(* CoDeSys 2.3 project: cy-22-wg-005.pro *)
(* Title: cy-22-wg - ClevergyAS *)
(* Libraries: Standard.lib 2.12.10 14:48:34, Util.lib 26.9.14 10:12:46, Visual.lib 2.12.10 14:48:34, WagoLibIdent.lib 25.2.13 11:12:16, WagoLibStatus.lib 2.12.10 14:48:32, SysLibFile.lib 2.12.10 14:48:34, SysLibRtc.lib 2.12.10 14:48:32, SysLibSockets.lib 10.2.11 09:20:54, SysLibEvent.lib 2.12.10 14:48:34, SysLibPlcCtrl.lib 2.12.10 14:48:32, SysLibCallback.lib 2.12.10 14:48:32, mod_com.lib 2.12.10 14:48:32, SerComm.lib 31.5.11 08:54:36, Serial_Interface_01.lib 22.4.13 12:50:14, Modb_l05.lib 22.4.13 12:50:12, WagoLibModbus_IP_01.lib 24.7.13 15:05:58 *)

(* PLC configuration (modules and I/O channels)
VPN_OUT2 AT %IX6.0 [BOOLOnX_I] Ch_1 Digital input
KEY_QE_ST AT %IX6.1 [BOOLOnX_I] Ch_2 Digital input
SCA01_1_DI AT %IX6.2 [BOOLOnX_I] Ch_3 Digital input
SCA01_2_DI AT %IX6.3 [BOOLOnX_I] Ch_4 Digital input
SCA01_3_DI AT %IX6.4 [BOOLOnX_I] Ch_5 Digital input
AT %IX6.5 [BOOLOnX_I] Ch_6 Digital input
AT %IX6.6 [BOOLOnX_I] Ch_7 Digital input
AT %IX6.7 [BOOLOnX_I] Ch_8 Digital input
DIG_TA1 AT %IW0 [WORDOnW_I] Ch_1 Input word
DIG_TA2 AT %IW1 [WORDOnW_I] Ch_2 Input word
0750-0653/0003-0000#03 RS485 Interface (Adjustable), 3 Bytes [Type_21_1_Channels] node 2, in %IB8 out %QB4 {INTTypePAAssignment = PLC; INTTypeModule = plugged}
  AT %IX2.0 [BOOLOnX_I] Transmission acknowledgement
  AT %IX2.1 [BOOLOnX_I] Reception request
  AT %IX2.2 [BOOLOnX_I] Initialization acknowledgement
  AT %IX2.3 [BOOLOnX_I] Input buffer is full
  AT %IX2.4 [BOOLOnX_I] Number of received characters Bit 0
  AT %IX2.5 [BOOLOnX_I] Number of received characters Bit 1
  AT %IX2.6 [BOOLOnX_I] Number of received characters Bit 2
  AT %IB5 [BYTEOnB_I] Input data Byte 0
  AT %IB6 [BYTEOnB_I] Input data Byte 1
  AT %IB7 [BYTEOnB_I] Input data Byte 2
  AT %QX0.0 [BOOLOnX_Q] Transmission request
  AT %QX0.1 [BOOLOnX_Q] Reception acknowledgement
  AT %QX0.2 [BOOLOnX_Q] Initialization request
  AT %QX0.4 [BOOLOnX_Q] Number of characters Bit 0
  AT %QX0.5 [BOOLOnX_Q] Number of characters Bit 1
  AT %QX0.6 [BOOLOnX_Q] Number of characters Bit 2
  AT %QB1 [BYTEOnB_Q] Output data Byte 0
  AT %QB2 [BYTEOnB_Q] Output data Byte 1
  AT %QB3 [BYTEOnB_Q] Output data Byte 2
0750-0653/0003-0000#03 RS485 Interface (Adjustable), 3 Bytes [Type_21_1_Channels] node 3, in %IB12 out %QB4 {INTTypePAAssignment = PLC; INTTypeModule = plugged}
  AT %IX4.0 [BOOLOnX_I] Transmission acknowledgement
  AT %IX4.1 [BOOLOnX_I] Reception request
  AT %IX4.2 [BOOLOnX_I] Initialization acknowledgement
  AT %IX4.3 [BOOLOnX_I] Input buffer is full
  AT %IX4.4 [BOOLOnX_I] Number of received characters Bit 0
  AT %IX4.5 [BOOLOnX_I] Number of received characters Bit 1
  AT %IX4.6 [BOOLOnX_I] Number of received characters Bit 2
  AT %IB9 [BYTEOnB_I] Input data Byte 0
  AT %IB10 [BYTEOnB_I] Input data Byte 1
  AT %IB11 [BYTEOnB_I] Input data Byte 2
  AT %QX2.0 [BOOLOnX_Q] Transmission request
  AT %QX2.1 [BOOLOnX_Q] Reception acknowledgement
  AT %QX2.2 [BOOLOnX_Q] Initialization request
  AT %QX2.4 [BOOLOnX_Q] Number of characters Bit 0
  AT %QX2.5 [BOOLOnX_Q] Number of characters Bit 1
  AT %QX2.6 [BOOLOnX_Q] Number of characters Bit 2
  AT %QB5 [BYTEOnB_Q] Output data Byte 0
  AT %QB6 [BYTEOnB_Q] Output data Byte 1
  AT %QB7 [BYTEOnB_Q] Output data Byte 2
LUX5_EN AT %QX4.0 [BOOLOnX_Q] Ch_1 Digital output
LUX6_EN AT %QX4.1 [BOOLOnX_Q] Ch_2 Digital output
LUX3_EN AT %QX4.2 [BOOLOnX_Q] Ch_1 Digital output
LUX4_EN AT %QX4.3 [BOOLOnX_Q] Ch_2 Digital output
LUX1_EN AT %QX4.4 [BOOLOnX_Q] Ch_1 Digital output
LUX2_EN AT %QX4.5 [BOOLOnX_Q] Ch_2 Digital output
Fieldbus variables [FB_VARS] node 1, in %IB0 out %QB0
Flag variables [FLAG_VARS] node 2, in %IB0 out %QB0
Modbus-Master [MB_MASTER] node 3, in %IB0 out %QB0
*)

(* Global variable list: Global_Constants *)
VAR_GLOBAL CONSTANT

	Plant_NAME			: STRING :='cySN:22 cyVER:0 - Coin OVS Curno';
	Plant_SN			: DWORD  :=22;	  	(* S/N Impianto di telecontrollo *)
	Plant_SW_VER		: WORD   :=0;		(* Versione SW installata *)

	(* Colour defines *)
	COLOR_RED			: DWORD	:= 16#2020F0;
	COLOR_YELLOW		: DWORD	:= 16#20F0F0;
	COLOR_GREEN			: DWORD	:= 16#20F020;
	COLOR_GREEN_OFF		: DWORD := 16#006000;

	(* Parameters *)
	Plant_DefaultTAmb	: INT	:=100;		(* [.1°C] Temperatura ambiente di default in caso di rottura sonda *)
	Plant_MaxRunTAmb	: INT   :=250; 		(* [.1°C] Temperatura ambiente massima funzionamento impianto *)
	Plant_AntiFreezeTAmb: INT   :=-40;		(* [.1°C] Antifreeze temperature, start circulators *)
	Plant_VRD_TAlarm	: INT   :=450; 		(* [.1°C] Temperatura di allarme VRD, blocco *)
	Plant_VRD_TMax		: INT   :=430; 		(* [.1°C] Setpoint massimo per uscita VRD *)
	Plant_VRD_TDefault	: INT	:=300;		(* [.1°C] Temperatura di default in caso di errore climatica *)
	Plant_CirOffDelay	: TIME	:=T#15m;	(* (Def.T#15m) Ritardo spegnimento pompe per ricircolo caldaia *)
	Plant_MaxWaterLoss	: WORD  :=2;		(* [lt/h] Massima perdita del circuito *)

	FeedbackTolerance	: WORD	:= 5;		(* 10% Tolerance on read measures *)

	(* Filesystem *)
	FilesPath  			: STRING :='S:\';

	(* TCP Logger *)
	Logger_SERVER		: STRING:='';
	Logger_IP			: STRING:='192.168.100.3';
	Logger_PORT			: WORD  :=80;
	Logger_GETSTART		: STRING:='GET /cygmsrv/hsgm.ashx?';
	Logger_GETEND		: STRING:='$R$N$R$N';
	Logger_CHECK		: STRING:='True';
	Logger_CRLF			: STRING:='$R$N';
	Logger_DataFile		: STRING:='S:\LOG.DAT';
	Logger_DataFileOld	: STRING:='S:\LOG.BCK';
	Logger_IndexFile	: STRING:='S:\LOG.IDX';
	Logger_ConnRetries	: BYTE:=5;
	Logger_RecoverMsgs	: BYTE:=25;

	(* TCP Remote *)
	Remote_PORT			: WORD  :=10;
	Remote_WELCOME		: STRING:='Connected$R$N';
	Remote_OK			: STRING:='OK$R$N';
	Remote_ERROR		: STRING:='ERROR$R$N';

	(* TCP Sockets *)
	MAX_SEND_TCP_SERVER					 : DWORD:=3000;(*60000*)
	MAX_RECEIVE_TCP_SERVER				 : DWORD:=3000;
	MAX_RECEIVE_TCP_SERVER_SOCKET	 	 : DWORD:=1500;
	MAX_SEND_TCP_CLIENT					 : DWORD:=3000;(*15000*)
	MAX_RECEIVE_TCP_CLIENT				 : DWORD:=1500;
	MAX_RECEIVE_TCP_CLIENT_SOCKET		 : DWORD:=1500;
	MAX_RECEIVE_UDP_SERVER				 : INT  :=1472;
	MAX_RECEIVE_UDP_CLIENT				 : INT  :=1472;
	CONNECT_WATCHDOG_TIME				 : TIME :=t#10s;

END_VAR

(* Global variable list: Global_Retain *)
VAR_GLOBAL RETAIN PERSISTENT
	Mode_Manual : BOOL := FALSE;

	Lux_ref	:	ARRAY [1..2,1..7] OF WORD;

	LuxWT	:	ARRAY [1..6] OF DWORD;	(* Lux working time non volatile counters *)
	LuxPOC	:	ARRAY [1..6] OF DWORD;	(* Lux power on cycles non volatile counters *)
END_VAR

(* Global variable list: Global_Variables *)
VAR_GLOBAL

	SYS    : typ_SYS;
	Logger : typ_Logger;
	CronEd : obj_CRON_EDITOR;

	(**** PLANT OBJECTS ****)
	CRON01 : obj_CRON		:= ( ID:=1 );		(* Controllo LUX01 *)
	CRON02 : obj_CRON		:= ( ID:=2 );		(* Controllo LUX02 *)
	CRON03 : obj_CRON		:= ( ID:=3 );		(* Controllo LUX03 *)
	CRON04 : obj_CRON		:= ( ID:=4 );		(* Controllo LUX04 *)
	CRON05 : obj_CRON		:= ( ID:=5 );		(* HVAC01 - Start Stop  *)
	CRON06 : obj_CRON		:= ( ID:=6 );		(* HVAC01 - Set Point raffreddamento *)
	CRON07 : obj_CRON		:= ( ID:=7 );		(* HVAC01 - Set Point riscaldamento *)
	CRON08 : obj_CRON		:= ( ID:=8 );		(* HVAC01 - ??? Set Point ECO Soglia Minima *)
	CRON09 : obj_CRON		:= ( ID:=9 );		(* HVAC01 - ??? Set Point ECO Soglia Massima *)
	CRON10 : obj_CRON		:= ( ID:=10 );		(* HVAC02 - Start Stop *)
	CRON11 : obj_CRON		:= ( ID:=11 );		(* HVAC02 - Set Point raffreddamento *)
	CRON12 : obj_CRON		:= ( ID:=12 );		(* HVAC02 - Set Point riscaldamento *)
	CRON13 : obj_CRON		:= ( ID:=13 );		(* HVAC02 - ??? Set Point ECO Soglia Minima *)
	CRON14 : obj_CRON		:= ( ID:=14 );		(* HVAC02 - ??? Set Point ECO Soglia Massima *)

	LUX01  : obj_LUXP		:= ( ID:=1, CTRL_MODE:=2, KEY_DEV:=FALSE );		(* Control mode: Scheduled -> Crono	*)
	LUX02  : obj_LUXP		:= ( ID:=2, CTRL_MODE:=2 );		(* Control mode: Scheduled -> Crono	*)
	LUX03  : obj_LUXP		:= ( ID:=3, CTRL_MODE:=0, KEY_DEV:=TRUE );		(* Control mode: Manual -> Switch *)
	LUX04  : obj_LUXP		:= ( ID:=4, CTRL_MODE:=2 );		(* Control mode: Scheduled -> Crono	*)
	LUX05  : obj_LUXP		:= ( ID:=5, CTRL_MODE:=2 );		(* Control mode: Scheduled -> Crono	*)
	LUX06  : obj_LUXP		:= ( ID:=6, CTRL_MODE:=1 );		(* Control mode: Automatic -> External device/sensor	*)

	AID01  : obj_ANALOG_IN_DIFF				:= (ID:=1, Lines:=3);
	AID02  : obj_ANALOG_IN_DIFF				:= (ID:=2, Lines:=3);

	MODB01 : obj_MODBUS						:= ( ID:=1 , COM:=2, BAUDRATE:=BAUD_9600, RS485:=TRUE );
	ANZ01  : obj_MODBUS_FRER_QUBOH			:= ( ID:=1 , Address:=1 );
	ANZ02  : obj_MODBUS_FRER_QUBOH			:= ( ID:=2 , Address:=2 );

	MODB02 : obj_MODBUS						:= ( ID:=2 , COM:=3, BAUDRATE:=BAUD_9600, RS485:=TRUE );
	HVAC01 : obj_HVAC_LENNOX_FGK190H2M_new	:= ( ID:=1 , ADDRESS:=1 );
	HVAC02 : obj_HVAC_LENNOX_FGK190H2M_new	:= ( ID:=2 , ADDRESS:=2 );

	MODB03 : obj_MODBUS_TCP					:= ( ID:=1,IP:='192.168.100.11');
	ZTHL01 : obj_ZTHL						:= ( ID:=1, Address:=2);
	ZTHL02 : obj_ZTHL						:= ( ID:=2, Address:=3);
	ZTHL03 : obj_ZTHL						:= ( ID:=3, Address:=5);
	ZTHL04 : obj_ZTHL						:= ( ID:=4, Address:=6);

	(**** SIMULATION ONLY ****)
(*	VPN_ST2		:BOOL:=TRUE;
	KEY_QE_ST	:BOOL:=TRUE;
*)

END_VAR

(* Data type in Logger *)
TYPE en_Logger_ErrLev :
(
	EL_Log			:=0,
	EL_Wrn			:=1,
	EL_Alarm			:=2,
	EL_AlarmStop		:=3
);
END_TYPE

(* Data type in Logger *)
TYPE en_Logger_Status :
(
	S_Logger_UNKNOWN := 0,
	S_Logger_IDLE,
	S_Logger_WAITCONN,
	S_Logger_WAITTX,
	S_Logger_WAITRESP,
	S_Logger_ERROR
);
END_TYPE

(* Data type *)
TYPE en_SYS_Objects :
(
	EO_SYS		:=0,  (* PLC *)
	EO_VPN		:=1,  (* VPN *)
	EO_DOOR	:=2,  (* Door & access control *)

	EO_CAL		:=10, (* Caldaia *)
	EO_CIR		:=11, (* Circolatore *)
	EO_CRON		:=12, (* Crono-termostato *)
	EO_VRD		:=13, (* Valvola miscelatore pannelli *)
	EO_CTL		:=14, (* Contalitri *)
	EO_CTB		:=15, (* Contabilizzatore *)
	EO_TPV		:=16, (* Temperature probes values *)
	EO_PPV		:=17, (* Pressure probes values *)
	EO_PBV		:=18, (* Over-Pressure Alarms *)
	EO_TBV		:=19, (* Over-Temperature Alarms *)
	EO_PMV		:=20, (* Under-Pressure Alarms *)
	EO_GRU		:=21, (* Gruppo termico *)
	EO_PDC		:=22, (* Pompa di calore *)
	EO_SOL		:=23, (* Pannello solare termico *)
	EO_ESOL		:=24, (* Pannello solare fotovoltaico *)
	EO_GAS		:=25, (* Contatore GAS *)
	EO_PORT		:=26, (* Misuratore di portata *)
	EO_FPV		:=27, (* Flow probes values *)
	EO_ANZ		:=28, (* Analizzatore di rete *)
	EO_SCA		:=29, (* Signal Control Alarms *)
	EO_LUX		:=30, (* Illumination point *)
	EO_LUXM		:=31, (* Metered illumination point*)
	EO_PSG		:=32, (* Sensore di passaggio *)
	EO_HVAC		:=33, (*Heating, Ventilating and Air Conditioning*)
	EO_HYGRV	:=34, (*Valori sensori di umidità relativa (0.1%)*)
	EO_COOV		:=35, (*Valori sensori CO2 (PPM)*)




	EO_ZGW			:=200,  (* ZigBee - Gateway *)
	EO_ZRM			:=201,	(* ZigBee - Repeater *)
	EO_ZREL			:=202,	(* ZigBee - Actuator rele *)
	EO_ZTHL			:=203,	(* ZigBee - Temperature Sensor *)

	EO_ASGW			:=250,	(* ASi - Gateway *)
	EO_ASCBI			:=251,	(* ASi - Input Board, Ciabatta *)

	EO_LON				:=1000, (* Bus - LON *)
	EO_MODBUS			:=1001, (* Bus - MODBUS *)
	EO_MBUS				:=1002, (* Bus - M-BUS *)
	EO_MODBUS_TCP	:=1003, (* Bus - MODBUS TCP *)

	EO_GENERIC			:=9000, (* Generic dataset *)
	EO_EXPO				:=9001 (* EXPO dataset *)
);
END_TYPE

(* Data type *)
TYPE en_SYS_Status :
(
	S_UNKNOWN  := 0,
	S_STARTUP,
	S_INIT_RTC,
	S_INIT_VAR,
	S_AUTOTEST,
	S_RUNNING,
	S_SHUTDOWN,
	S_HALT
);
END_TYPE

(* Data type in Plant_Objects *)
TYPE typ_Condition :
STRUCT
	Enable		:	BYTE;	(*	0: Condition event not used		(disable condition event)
								1: Boolean event: trig On	(rele, switch, sensors digital input..)
								2:    ''    ''  : trig Off		
								3:	  ''    ''  : trig On/Off
								4: Tod event: trig On		(Time of day)
								5: Tod event: trig Off		(Trig On/Off not expected -> it's a schedule! )
							 *)

	(* Boolean event *)
	OnIN		:	BOOL;	(* Input event generating an On *)
	OffIN		:	BOOL;	(* Input event generating an Off  *)

	OnValue		:	BOOL;	(* Value to trig an On *)
	OffValue	:	BOOL;	(*   ''        ''   Off	 *)


	(* Time of the day event (absolute time) *)
	OnTime		:	TOD;	(* Time at which trig an On (hh:mm) *)
	OffTime		:	TOD;	(*  ''            ''     Off (hh:mm)  *)


END_STRUCT
END_TYPE

(* Data type in Plant_Objects *)
TYPE typ_Cron_Calendar :
STRUCT
	Profile		: ARRAY[0..384] OF BYTE;
END_STRUCT
END_TYPE

(* Data type in Plant_Objects *)
TYPE typ_Cron_Jolly :
STRUCT
	Start		: DT;
	End			: DT;
	Temp		: WORD;
	Flags		: WORD; (* B0:Enabled B1..B15:Unused *)
END_STRUCT
END_TYPE

(* Data type in Plant_Objects *)
TYPE typ_Cron_Profile :
STRUCT
	Flags		: WORD;
	Setpoint	: ARRAY [0..95] OF WORD;
END_STRUCT
END_TYPE

(* Data type in Logger *)
TYPE typ_Logger :
STRUCT
	Status		: en_Logger_Status;

	SendReq		: BOOL;
	SendIdx		: DWORD;
	SendData	: ARRAY [0..MAX_SEND_TCP_CLIENT] OF BYTE;
	SendLen		: DINT;

	TData		: ARRAY [0..MAX_SEND_TCP_CLIENT] OF BYTE;
	TLen		: DINT;

	LastIdxPos	: DWORD;

	(* Temporary variables used by objects *)
	s1			: STRING(256);
	i1			: WORD;

END_STRUCT
END_TYPE

(* Data type in Plant_Objects *)
TYPE typ_MODBUS_ABB_DMTME72 :
STRUCT
	V_3P		: DWORD; (* V *)
	V_L1N		: DWORD;
	V_L2N		: DWORD;
	V_L3N		: DWORD;
	V_L1L2		: DWORD;
	V_L2L3		: DWORD;
	V_L3L1		: DWORD;
	I_3P		: DWORD; (* 10^-3 A *)
	I_L1		: DWORD;
	I_L2		: DWORD;
	I_L3		: DWORD;
	PF_3P		: DINT;	 (* 10^-3 *)
	PF_L1		: DINT;
	PF_L2		: DINT;
	PF_L3		: DINT;
	COS_3P		: DINT;  (*NO!*)
	COS_L1		: DINT;
	COS_L2		: DINT;
	COS_L3		: DINT;
	VA_3P		: DWORD; (* VA *)(*NO!*)
	VA_L1		: DWORD;
	VA_L2		: DWORD;
	VA_L3		: DWORD;
	P_3P		: DWORD; (* W *)
	P_L1		: DWORD;
	P_L2		: DWORD;
	P_L3		: DWORD;
	Q_3P		: DWORD; (* VAr *)
	Q_L1		: DWORD;
	Q_L2		: DWORD;
	Q_L3		: DWORD;

	WH_3P		: DWORD; (* 10^-1 kWh *)
	VARH_3P		: DWORD; (* 10^-1 kVArh *)
	FREQ		: DWORD; (* 10^-3 Hz *)

	I_L1_Max	: DWORD;
	I_L2_Max	: DWORD;
	I_L3_Max	: DWORD;
	P_3P_Max	: DWORD;
	Q_3P_Max	: DWORD;
	P_3P_Avg15m	: DWORD;

END_STRUCT
END_TYPE

(* Data type in Plant_Objects *)
TYPE typ_MODBUS_FRER_QUBOH :
STRUCT
	V_L1N		:	DWORD;	(* E-3 V *)
	V_L2N		:	DWORD;
	V_L3N		:	DWORD;
	V_L1L2		:	DWORD;
	V_L2L3		:	DWORD;
	V_L3L1		:	DWORD;
	I_L1		:	DWORD;	(* E-3 A *)
	I_L2		:	DWORD;
	I_L3		:	DWORD;

	FREQ		:	DWORD;	(* E-3 Hz *)

	P_3P		:	DWORD;	(* W *)
	Q_3P		:	DWORD;	(* VAr *)
	PF_3P		:	DINT;	(* E-3 *)
	WH_3P		:	DWORD;	(* Wh *)
	VARH_3P		:	DWORD;	(* VArh *)
	Multiplier	:	DWORD;

	V_3P		:	DWORD;	(* E-3 V *)
	I_3P		:	DWORD;	(* E-3 A *)

	COS_3P		:	DINT;	(* E-3 *)

	VA_3P		:	DWORD;	(* VA *)
	P_L1		:	DWORD;	(* W *)
	P_L2		:	DWORD;
	P_L3		:	DWORD;
	Q_L1		:	DWORD;	(* VAr *)
	Q_L2		:	DWORD;
	Q_L3		:	DWORD;
	VA_L1		:	DWORD;	(* VA *)
	VA_L2		:	DWORD;
	VA_L3		:	DWORD;
	PF_L1		:	DINT;	(* E-3 *)
	PF_L2		:	DINT;
	PF_L3		:	DINT;
	COS_L1		:	DINT;	(* E-3 *)
	COS_L2		:	DINT;
	COS_L3		:	DINT;

	P_3P_Max	:	DWORD;	(* W *)
	P_3P_Avg	:	DWORD;

	I_L1_Max	:	DWORD;	(* E-3 A *)
	I_L2_Max	:	DWORD;
	I_L3_Max	:	DWORD;

	Q_3P_Max	:	DWORD;	(* VAr *)

END_STRUCT
END_TYPE

(* Data type in Plant_Objects *)
TYPE typ_MODBUS_HVAC_LENNOX_FGK190H2M :
STRUCT


(* valori da scrivere *)

	Heartbeat						:WORD;	(*holding registers 1 *)
	SP_Raffreddamento			:WORD;	(*holding registers 2 *)
	SP_Riscaldamento			:WORD;	(*holding registers 3 *)


	TempAmbienteBMS			:INT;	(*holding registers 20 *)
	UmiditaAmbienteBMS		:INT;	(*holding registers 21 *)
	TempEsternaBMS				:INT;	(*holding registers 22 *)
	UmiditaEsternaBMS			:INT;	(*holding registers 23 *)

	On_Off_Unita					:WORD;    (* holding registers  84 *)

	SP_MinPortataAriaECO		:WORD;	(*holding registers 187 *)
	SP_MAXPortataAriaECO		:WORD;	(*holding registers 188 *)


(* valori da Leggere *)


	ErrorCode						:WORD;	(*holding registers 36 *)
	TempAmbiente				:INT;	(*holding registers 37 *)
	TempEserno					:INT;	(*holding registers 38 *)
	TempMandata					:INT;	(*holding registers 39 *)
	TempRipresa					:INT;	(*holding registers 40 *)
	RelUmiditaAmbiente			:INT;	(*holding registers 41 *)
	AbsUmiditaAmbiente			:INT;	(*holding registers 42 *)
	RelUmiditaEsterno			:INT;	(*holding registers 43 *)
	AbsUmiditaEsterno			:INT;	(*holding registers 44 *)
	PressDiff						:INT;	(*holding registers 45 *)
	LivCO2						:INT;	(*holding registers 46 *)
	ApValvAria						:INT;	(*holding registers 47 *)
	ApValvGAS						:INT;	(*holding registers 48 *)
	ResElettrica					:INT;	(*holding registers 49 *)
	ApValvAcquaCalda			:INT;	(*holding registers 50 *)
	PercUmidificatore				:INT;	(*holding registers 51 *)

	h_VentSoffiante			:DWORD;	(*holding registers 62 *)
(*	h_VentSoffiante_h				:WORD;	(*holding registers 63 *)*)
	h_Compressore1			:DWORD;	(*holding registers 64 *)
(*	h_Compressore1_h			:WORD;	(*holding registers 65 *)*)
	h_Compressore2			:DWORD;	(*holding registers 66 *)
(*	h_Compressore2_h			:DWORD;	(*holding registers 67 *)*)
	h_Compressore3			:DWORD;	(*holding registers 68 *)
(*	h_Compressore3_h			:DWORD;	(*holding registers 69 *) *)
	h_Compressore4			:DWORD;	(*holding registers 70 *)
(*	h_Compressore4_h			:WORD;	(*holding registers 71 *) *)

	bit_Allarme01					:WORD;	(*holding registers 74 *)
	bit_Allarme02					:WORD;	(*holding registers 75 *)
	bit_Allarme03					:WORD;	(*holding registers 76 *)
	bit_Allarme04					:WORD;	(*holding registers 77 *)
	bit_Allarme05					:WORD;	(*holding registers 78 *)
	bit_Allarme06					:WORD;	(*holding registers 79 *)
	bit_Allarme07					:WORD;	(*holding registers 80 *)


(*
	SP_Umidificatore				:WORD;	(*holding registers 07H *)
	SP_Deumidificatore			:WORD;	(*holding registers 08H *)

*)

END_STRUCT
END_TYPE

(* Data type in Plant_Objects *)
TYPE typ_MODBUS_HVAC_LENNOX_FGK190H2M_new :
STRUCT

	BoolStatus		:	WORD;

	AlarmCode		:	WORD;
	Tenv			:	INT;	(* Environment temperature	[.1 °C]	*)
	Text			:	INT;	(* External temperature [.1 °C]	*)
	Tsend			:	INT;	(* Send temperature [.1 °C]		*)
	Treturn			:	INT;	(* Retrun temperature [.1 °C]	*)
	RH_env			:	WORD;	(* Environment relative humidity [.1 %]	*)
	AH_env			:	WORD;	(* Environment absolute humidity [.1 g/Kg]	*)
	RH_ext			:	WORD;	(* External relative humidity [.1 %]	*)
	AH_ext			:	WORD;	(* External absolute humidity [.1 g/Kg]	*)
	AirDiffPressure	:	WORD;	(* Differential air pressure [Pa]	*)
	CO2_ppm			:	WORD;	(* [ppm]	*)
	AirValve		:	WORD;	(* [%]	*)
	AirGas			:	WORD;	(* [%]	*)
	Triac			:	WORD;	(* Electrical heaters [%]	*)
	HWB				:	WORD;	(* Hot water battery [%]	*)
	Humidifier		:	WORD;	(* [%]	*)

	HourVent		:	DWORD;	(* Blow ventilator working hours [h]	*)
	HourCir1Comp1	:	DWORD;	(* Circuit 1 Compressor 1 working hours [h]	*)
	HourCir1Comp2	:	DWORD;	(* Circuit 1 Compressor 2 working hours [h]	*)
	HourCir2Comp1	:	DWORD;	(* Circuit 2 Compressor 1 working hours [h]	*)
	HourCir2Comp2	:	DWORD;	(* Circuit 2 Compressor 2 working hours [h]	*)

	Alarm1			:	WORD;
	Alarm2			:	WORD;
	Alarm3			:	WORD;
	Alarm4			:	WORD;
	Alarm5			:	WORD;
	Alarm6			:	WORD;
	Alarm7			:	WORD;

END_STRUCT
END_TYPE

(* Data type in Plant_Objects *)
TYPE typ_MODBUS_VAR : (* Gestione parametri MODBUS *)
STRUCT
	SlaveAddress		: BYTE;
	FunCode				: BYTE;
	FunAddress			: WORD;
	Refresh_Time		: BYTE; (* 0:No refresh x:Refresh in seconds *)
	Refresh_Cnt			: BYTE; (* INTERNAL *)
	Variable			: POINTER TO WORD;
	Variable_Size		: BYTE;
	Variable_Mirror 	: WORD; (* INTERNAL [Force refresh on read variables when <>0] *)
END_STRUCT
END_TYPE

(* Data type *)
TYPE typ_SYS :
STRUCT
	Status			: en_SYS_Status;
	Warning			: BOOL;
	Alarm			: BOOL;
	AlarmStop		: BOOL;

	Time_LogString	: STRING;
	Time_Year		: WORD;
	Time_Month		: BYTE;
	Time_Day		: BYTE;

	Time_CT_DT		: DT;
	Time_CT_Day		: WORD;
	Time_CT_Quarter	: BYTE;

	LastLogs_Idx	: BYTE;
	LastLogs_Dat	: ARRAY[0..5] OF STRING;
	LastLogs_Msg	: ARRAY[0..5] OF STRING;

END_STRUCT
END_TYPE

(* POU PLC_PRG, ST *)
PROGRAM PLC_PRG
VAR
	Timer1: TON; (* Fast controls tick *)
	Timer2: TON; (* Plant control tick *)
	Timer3: TON; (* Logger timer *)
	SetPointTempAmbiente: INT;
	Temperatura1: INT;
	Temperatura2: INT;
	SetPointTempEsterna: INT;
END_VAR
(******************************************************************************
 ****                           MAIN TASK CODE                             ****
 ******************************************************************************

	Network setup:
		IP  = 192.168.100.2 | MSK = 255.255.255.0
		GW	= 192.168.100.1 | DNS = 192.168.100.1
		SNTP = 193.204.114.232 (3600s) ==> 192.168.100.3

*)

(*==============================*)
(*===== Main status machine ====*)
(*==============================*)
Main_Stm();

(*==============================*)
(*== Running cycle operations ==*)
(*==============================*)
IF SYS.Status>S_INIT_VAR THEN

	(* Execute MODBUS process *)
	MODB01();
	ANZ01(ModBus:=MODB01);
	ANZ02(ModBus:=MODB01);

	(* Execute MODBUS process *)
	MODB02();
	HVAC01(MODBUS:=MODB02);
	HVAC02(MODBUS:=MODB02);

	(* Execute MODBUS process *)
	MODB03();
	(* Zigbee temeprature probes *)
	ZTHL01(ModBus:=MODB03);
	ZTHL02(ModBus:=MODB03);
	ZTHL03(ModBus:=MODB03);
	ZTHL04(ModBus:=MODB03);

	(* Execute feedback *)
	AID01( AdcValue:=DIG_TA1, Out1=>LUX1_EN, Out2=>LUX2_EN, Out3=>LUX3_EN );
	AID02( AdcValue:=DIG_TA2, Out1=>LUX4_EN, Out2=>LUX5_EN, Out3=>LUX6_EN );

END_IF

(*==============================*)
(*== System cycle operations ===*)
(*==============================*)
(* Execute TCP processes *)
Logger_Proc();
Remote_Proc();
(* Update user led *)
USRLED_Update();
(* Execute Cron Editor commands *)
CronEd();

(**** SIMULATION ONLY ****)
(*...*)
END_PROGRAM
ACTION Main_Stm:
CASE Sys.Status OF

	S_STARTUP:
		Sys.Status:=S_INIT_RTC;

	S_INIT_RTC:
		(* Check RTC and update from network *)
		RTC_Update();
		(* Check time *)
		IF Sys.Time_Year>2000 THEN
			Sys.Status:=S_INIT_VAR;
		END_IF

	S_INIT_VAR:
		LogEv(EL_Wrn,EO_SYS,0,1,CONCAT('System_startup_v',WORD_TO_STRING(Plant_SW_VER)));

		(* Conditional settings for LUXs *)
		LUX01.CTRL_COND.Enable := 0;
		LUX02.CTRL_COND.Enable := 0;
		LUX03.CTRL_COND.Enable := 0;
		LUX04.CTRL_COND.Enable := 0;
		LUX05.CTRL_COND.Enable := 0;
		LUX06.CTRL_COND.Enable := 5;
		LUX06.CTRL_COND.OffTime:= TOD#21:00;
		LUX06.CTRL_COND.OnTime := TOD#08:00;

		Sys.Status:=S_RUNNING;

	S_RUNNING:
		Timer1(IN:=NOT Timer1.Q,PT:=T#50ms);
		IF Timer1.Q THEN
			(* Update meters *)

			(* Update system checks *)
			SYS_Proc();
		END_IF

		Timer2(IN:=NOT Timer2.Q,PT:=T#500ms);
		IF Timer2.Q THEN
			(* Read current date/time *)
			RTC_Update();
			(* Execute plant operations *)
			(* LUX cronos *)
			CRON01();
			CRON02();
			CRON03();
			CRON04();
			(* HVAC cronos *)
			CRON05();
			CRON06();
			CRON07();
			CRON08();
			CRON09();
			CRON10();
			CRON11();
			CRON12();
			CRON13();
			CRON14();

			LUX01(CTRL_KEY:=SCA01_1_DI, CTRL_CRON:=INT_TO_BOOL(CRON01.SetPoint),
				  WORKINGTIME:=LuxWT[1], POWERONCYCLES:=LuxPOC[1],
				  OUT_EN=>AID01.In1, OUT_ST:=AID01.Alarm);
			LUX02(CTRL_CRON:=INT_TO_BOOL(CRON02.SetPoint),
				  WORKINGTIME:=LuxWT[2], POWERONCYCLES:=LuxPOC[2],
				  OUT_EN=>AID01.In2, OUT_ST:=AID01.Alarm);
			LUX03(CTRL_KEY:=SCA01_3_DI,
				  WORKINGTIME:=LuxWT[3], POWERONCYCLES:=LuxPOC[3],
				  OUT_EN=>AID01.In3, OUT_ST:=AID01.Alarm);
			LUX04(CTRL_CRON:=INT_TO_BOOL(CRON03.SetPoint),
				  WORKINGTIME:=LuxWT[4], POWERONCYCLES:=LuxPOC[4],
				  OUT_EN=>AID02.In1, OUT_ST:=AID02.Alarm);
			LUX05(CTRL_CRON:=INT_TO_BOOL(CRON04.SetPoint),
				  WORKINGTIME:=LuxWT[5], POWERONCYCLES:=LuxPOC[5],
				  OUT_EN=>AID02.In2, OUT_ST:=AID02.Alarm);
			LUX06(CTRL_EXT_DS:=SCA01_2_DI,
				  WORKINGTIME:=LuxWT[6], POWERONCYCLES:=LuxPOC[6],
				  OUT_EN=>AID02.In3, OUT_ST:=AID02.Alarm);

			(* Start measurement *)
			AID01.Measure();
			AID02.Measure();

			(* scelta del set point *)
			Temperatura1 := SEL(ZTHL01.ERR,ZTHL01.OUT_TEMP,ZTHL02.OUT_TEMP);
			Temperatura2 :=	SEL(ZTHL02.ERR,ZTHL02.OUT_TEMP,ZTHL01.OUT_TEMP);

			HVAC01(
					SetPointColdDay:=CRON06.SetPoint ,
					SetPointHeatDay:=CRON07.SetPoint ,
					SetBmsTenv:=(Temperatura1+Temperatura2)/2 ,
					SetBmsRHenv:= ,
					SetBmsText:= ,
					SetBmsRHext:= ,
					OnOff:= INT_TO_BOOL(CRON05.SetPoint) ,
					MinThrECO:=CRON08.SetPoint ,
					MaxThrECO:=CRON09.SetPoint ,
					modBus:=MODB02,
					 );

			(* scelta del set point *)
			Temperatura1 := SEL(ZTHL03.ERR,ZTHL03.OUT_TEMP,ZTHL04.OUT_TEMP);
			Temperatura2 :=	SEL(ZTHL04.ERR,ZTHL04.OUT_TEMP,ZTHL03.OUT_TEMP);

			HVAC02(
					SetPointColdDay:=CRON11.SetPoint ,
					SetPointHeatDay:=CRON12.SetPoint ,
					SetBmsTenv:=(Temperatura1 +Temperatura2)/2 ,
					SetBmsRHenv:= ,
					SetBmsText:= ,
					SetBmsRHext:= ,
					OnOff:= INT_TO_BOOL(CRON10.SetPoint) ,
					MinThrECO:=CRON13.SetPoint ,
					MaxThrECO:=CRON14.SetPoint ,
					modBus:=MODB02,
					 );

				(* Test toggle *)
			(*	IF TEST1 THEN TEST1:=FALSE; ELSE TEST1:=TRUE; END_IF   *)
		END_IF

		Timer3(IN:=NOT Timer3.Q,PT:=T#5m);
		IF Timer3.Q THEN
			(* Trig logger *)
			LogTrig();
			(* Execute temporary CSV logger *)
			(*CSV_Log();*)
		END_IF

	S_SHUTDOWN:
		(* Stop sistema *)
		Sys.Status:=S_STARTUP;

	S_HALT:
		(* Aspetta uscita manuale *)
		Sys.Status:=S_STARTUP;

ELSE
	Sys.Status:=S_STARTUP;
END_CASE;
END_ACTION

(* POU TCP_Logger/Logger_Proc, ST *)
PROGRAM Logger_Proc
VAR
	c1:         	TCPCLIENT;

	Open:	    	BOOL;
	IpAddr:			DWORD;
	InetAddr:		DWORD;
	Connected:  	BOOL;
	Error:      	DINT;
	TxTrig:     	BOOL;
	RxData:			ARRAY [0..MAX_RECEIVE_TCP_CLIENT] OF BYTE;
	RxLen:			DINT;

	Retry:			BYTE;	(* Counter for connection retries *)
	Recovered:		BYTE;	(* Counter for recovered unsent messages *)

	i:				DINT;
	pos:			DWORD;
	hFile:			DWORD;

END_VAR
(*=== State machine ===*)
CASE Logger.Status OF

	S_Logger_UNKNOWN:
		(* Startup *)
		Logger.SendReq:=FALSE;
		Open:=FALSE;
		Logger.Status:=S_Logger_IDLE;

	S_Logger_IDLE:
		(* Wait request *)
		IF Logger.SendReq THEN
			(* Resolve server name or use static IP *)
			IF LEN(Logger_SERVER)=0 THEN
				InetAddr:=SysSockInetAddr(Logger_IP);
			ELSE
				IpAddr:=SysSockGetHostByName(ADR(Logger_SERVER));
				DWORDSWAP(pIn:=ADR(IpAddr), pOut:=ADR(InetAddr));
			END_IF
			TxTrig:=FALSE;
			RxLen:=0;
			(* Open connection *)
			Open:=TRUE;
			Logger.Status:=S_Logger_WAITCONN;
		END_IF

	S_Logger_WAITCONN:
		(* Wait connection *)
		IF Connected THEN
			(* Send data *)
			TxTrig:=TRUE;
			Logger.Status:=S_Logger_WAITTX;
		END_IF
		IF Error>0 THEN
			Open:=FALSE;
			Logger.Status:=S_Logger_ERROR;
		END_IF

	S_Logger_WAITTX:
		(* Wait transmission *)
		IF NOT TxTrig THEN
			Logger.Status:=S_Logger_WAITRESP;
		END_IF
		IF Error>0 THEN
			Open:=FALSE;
			Logger.Status:=S_Logger_ERROR;
		END_IF

	S_Logger_WAITRESP:
		(* Wait response *)
		IF Connected=FALSE (* OR TIMEOUT!! *) THEN
			Open:=FALSE;
			(* Check response *)
			IF RxLen>=4 AND CHKSTRING(pString:=ADR(RxData), pPattern:=ADR(Logger_CHECK)) THEN
				Logger.SendReq:=FALSE;
				Retry:=0;
				(* Check unsent messages to flush *)
				IF Recovered<Logger_RecoverMsgs THEN
					MsgChk();
					IF Logger.SendReq=TRUE THEN
						Recovered:=Recovered+1;
					ELSE
						Recovered:=0;
					END_IF
				ELSE
					Recovered:=0;
				END_IF
				Logger.Status:=S_Logger_IDLE;
			ELSE
				Logger.Status:=S_Logger_ERROR;
			END_IF
		END_IF

	S_Logger_ERROR:
		(* Connection error or send failure *)
		Retry:=Retry+1;
		IF Retry>Logger_ConnRetries THEN
			(* Save message as unsent *)
			MsgSave();
			Logger.SendReq:=FALSE;
			Retry:=0;
		END_IF
		Logger.Status:=S_Logger_IDLE;

ELSE
	Logger.Status:=S_Logger_UNKNOWN;
END_CASE


(*=== Execute client lib ===*)
c1(
	xOpenConnection			:= Open,
	dwInetAddr 				:= InetAddr,
	wPortNumber				:= Logger_PORT,
	ptSendData				:= ADR(Logger.SendData),
	diSendCount				:= Logger.SendLen,
	tConnectWatchdogTime	:= t#10s,
	xStartSend				:= TxTrig,
	aReceiveBuffer			:= RxData,
	diReceiveCount			:= RxLen,
	xConnected				=> Connected,
	diError					=> Error
);

(*=== Process Rx data ===*)
(*IF RxLen>0 THEN
	RxLen:=0;
END_IF*)
END_PROGRAM
ACTION MsgChk:
(* Open index file *)
hFile:=SysFileOpen(Logger_IndexFile,'r');
IF hFile=0 THEN
	RETURN;
END_IF
(* Search oldest message to recover *)
SysFileSetPos(hFile,Logger.LastIdxPos);
Logger.SendLen:=0;
REPEAT
	SysFileRead(hFile, ADR(Logger.SendIdx), SIZEOF(Logger.SendIdx));
	pos:=SysFileGetPos(hFile);
	SysFileRead(hFile, ADR(Logger.SendLen), SIZEOF(Logger.SendLen));
UNTIL
	SysFileEOF(hFile) OR Logger.SendLen<>0
END_REPEAT
SysFileClose(hFile);
(* Delete index file when all messages are recovered *)
IF Logger.SendLen=0 THEN
	Logger.LastIdxPos:=0;
	SysFileDelete(Logger_IndexFile);
	RETURN;
END_IF
(* Recover message data *)
hFile:=SysFileOpen(Logger_DataFile,'r');
IF hFile<>0 THEN
	SysFileSetPos(hFile,Logger.SendIdx);
	SysFileRead(hFile,ADR(Logger.SendData),Logger.SendLen);
	Logger.SendReq:=TRUE;
	SysFileClose(hFile);
END_IF
(* Clear index entry *)
hFile:=SysFileOpen(Logger_IndexFile,'a');
IF hFile<>0 THEN
	SysFileSetPos(hFile,pos);
	i:=0;
	SysFileWrite(hFile, ADR(i), 4);
	Logger.LastIdxPos:=SysFileGetPos(hFile);
	SysFileClose(hFile);
END_IF
END_ACTION
ACTION MsgSave:
(* Add log position in recovery indexes *)
hFile:=SysFileOpen(Logger_IndexFile,'a');
SysFileWrite(hFile, ADR(Logger.SendIdx), SIZEOF(Logger.SendIdx));
SysFileWrite(hFile, ADR(Logger.SendLen), SIZEOF(Logger.SendLen));
SysFileClose(hFile);
END_ACTION

(* POU Utils Functions/TCPCLIENT, ST *)
FUNCTION_BLOCK TCPCLIENT
(***********************************************************************************************************	*)
(* Version: 1.3b                        			          													*)
(* Date: 28.10.2014                   				          							            			*)
(***********************************************************************************************************	*)
(* WAGO Kontakttechnik GmbH Hansastr. 27 32423 Minden(Westf.)													*)
(* Tel. +0049 571/887-0 Fax. +0049 571/887-0																	*)
(* Author: VB																									*)
(***********************************************************************************************************	*)
(*Description:	A TCP client to read and write data with additional connection watchdog							*)
(*History:																										*)
(*Version 1.3b: 28.10.2014: Use DWORD address for IP (Andrea Ravasio)											*)
(*Version 1.3: 11.02.2011: Changes according to 750-880/881											 			*)
(*Version 1.2: 29.08.2007 Bugfix TCP Client																		*)
(*Version 1.1: 15.01.2007 Changes according to FW11																*)
(*Version 1.0: 09.03.2006 Release																				*)
(***********************************************************************************************************	*)
VAR CONSTANT
	STATE_CREATE     				 : BYTE:= 0;
	STATE_OPEN     					 : BYTE:= 1;
	STATE_IOCTL    					 : BYTE:= 2;
	STATE_CONNECT     				 : BYTE:= 10;
	STATE_TX       					 : BYTE:= 20;
	STATE_RX       					 : BYTE:= 30;
	STATE_CLOSE    					 : BYTE:= 40;
	STATE_ERROR_TRAP			     : BYTE:= 200;
END_VAR

VAR_INPUT
	xOpenConnection					: BOOL;
	dwInetAddr						: DWORD; (* <== Use SysSockInetAddr() value or
													swapped bytes order of SysSockGetHostByName() value *)
	wPortNumber						: WORD;
	ptSendData						: POINTER TO ARRAY[0..MAX_SEND_TCP_CLIENT] OF BYTE;
	diSendCount						: DINT;
	tConnectWatchdogTime		    : TIME := t#10s;
END_VAR
VAR_OUTPUT
	xConnected						: BOOL;
	diError 						: DINT := 0;
END_VAR
(* ErrorCodes -----------------------------------------
	16#8001 => No socket descriptor available 
	16#8002 => SysSockSend returns -1 
	16#8003 => Socket was "gracefully closed" 
	16#8004 => switching to none blocking mode fails
	16#8005 => SysSockClose() returns FALSE 
    16#8006 => SysSockConnect() fails
    16#8007 => SysSockSend() fails
	16#8008 => error state machine 
	16#8009 => timeout while waiting for data from server 
------------------------------------------------------------*)
VAR_IN_OUT
	xStartSend							: BOOL;
	aReceiveBuffer						: ARRAY [0..MAX_RECEIVE_TCP_CLIENT] OF BYTE;
	diReceiveCount						: DINT;
END_VAR
VAR
	m_State								: BYTE := 0;
	m_ReceiveBuffer						: ARRAY [0..MAX_RECEIVE_TCP_CLIENT_SOCKET] OF BYTE;
	m_Socket							: DINT;
	m_AddressInfo						: SOCKADDRESS;
	m_BytesReceived						: DINT;
	m_diReturn							: DINT;
	m_xReturn							: BOOL;
	m_IoCtlParameter  					: DINT := 1; (* IOCTL-Parameter for non-blocking mode of sockets *)
	i									: INT;
	T_Connect							: TON;
	m_count								: DINT;
	diOption							: DINT := 1;
	m_Blocking   						: DINT := 0;
END_VAR
IF xOpenConnection THEN
	(* State maschine *)
	CASE  m_State OF

	(* -------------------------------------------------------------------------*)
	STATE_CREATE:
			(* create socket descriptor*)
			m_Socket := SysSockCreate(diAddressFamily	:= SOCKET_AF_INET,
													 diType		:= SOCKET_STREAM,
													 diProtocol := SOCKET_IPPROTO_TCP);
			IF m_Socket >= 0 THEN
			(*Set Push-Bit*)
				IF ADR(%MW0)=16#30000000  OR ADR(%MW0)=16#20000000 THEN (*841 or 881*)
					SysSockSetOption(
						diSocket:=m_Socket,
						diLevel:=6,
						diOption:=SOCKET_TCP_NODELAY,
						pOptionValue:=ADR(diOption),
						diOptionLength:=SIZEOF(diOption));
				ELSE
						;
				END_IF
				m_State := STATE_IOCTL; (* succesful *)
			ELSE
				diError := 16#8001;  (* no socket descriptor available *)
				m_State := STATE_ERROR_TRAP;
			END_IF

	(* -------------------------------------------------------------------------*)
	STATE_IOCTL: (* change  socket mode  to none blocking *)
		m_diReturn := SysSockIoctl( m_Socket, SOCKET_FIONBIO, ADR(m_IoCtlParameter));
		IF m_diReturn <> 0 THEN
			m_AddressInfo.sin_family := SOCKET_AF_INET;
			m_AddressInfo.sin_port := SysSockNtohs(wPortNumber);
			m_AddressInfo.sin_addr := dwInetAddr;
			m_State := STATE_CONNECT;
		ELSE
			diError := 16#8004;  (* switching to none blocking mode fails *)
			m_State := STATE_ERROR_TRAP;
		END_IF


	(* -------------------------------------------------------------------------*)
	STATE_CONNECT: (* connect with server *)
		T_Connect(IN:=TRUE , PT:=tConnectWatchdogTime);(*activate watchdog for establishing connection to a server*)
		m_xReturn := SysSockConnect ( m_Socket, ADR(m_AddressInfo),  SIZEOF(m_AddressInfo));
		IF m_xReturn THEN (* succesful *)
			IF xStartSend THEN
				m_State := STATE_TX;(*transmit data*)
			ELSE
				m_State := STATE_RX;(*wait for data from server*)
			END_IF
			xConnected:=TRUE;
			T_Connect(IN:=FALSE);
		ELSE
			IF T_Connect.Q THEN
				diError := 16#8006;  (* connect fails *)
				xConnected:=FALSE;
				T_Connect(IN:=FALSE);
				m_State := STATE_ERROR_TRAP;
				SysSockClose( m_Socket);
			ELSE
				m_State := STATE_CONNECT;(*client still  tries to set up connection*)
			END_IF
		END_IF


	STATE_TX:	 (* send TCP-message *)
		m_diReturn := SysSockSend(diSocket := m_Socket,
								  pbyBuffer := ADR(ptSendData^[0]),
								  diBufferSize := diSendCount-m_count,
								  diFlags := 0);

		CASE m_diReturn OF
		-1:	(* ERROR *)
			T_Connect(IN:=TRUE , PT:=CONNECT_WATCHDOG_TIME);(*activate watchdog to check communication*)
			IF t_Connect.Q THEN
				diError := 16#8007;
				T_Connect(IN:=FALSE);
				m_State:=STATE_CLOSE;
			END_IF
		0: (* socket was "gracefully closed" *)
			m_State := STATE_CLOSE;
			diError := 16#8003;
		ELSE (* succesful *)
			m_count:=m_count+m_diReturn;
			IF m_count>=diSendCount THEN
				diError := 16#0000;
				m_State := STATE_RX;
				m_count:=0;
				xStartSend:=FALSE;
			END_IF
			T_Connect(IN:=FALSE);
		END_CASE

	(* -------------------------------------------------------------------------*)
	STATE_RX: (* process receive data *)
			m_BytesReceived := SysSockRecv(	diSocket 	:= m_Socket,
										pbyBuffer 	:= ADR(m_ReceiveBuffer),		(* Address of receive buffer *)
										diBufferSize:= SIZEOF(m_ReceiveBuffer),
										diFlags		:= 0);

			CASE m_BytesReceived OF
			-1:	(* No data available or error occured *)
				T_Connect(IN:=TRUE , PT:=tConnectWatchdogTime);(*activate watchdog to check communication*)
				IF t_Connect.Q THEN
					diError:=16#8009;
					T_Connect(IN:=FALSE);
					m_State:=STATE_CLOSE;
				END_IF
				IF xStartSend THEN
					m_State:=STATE_TX	;(* WAIT IN THIS STATE  and check for arriving data or new send command*)
				END_IF;
			0: (* socket was "gracefully closed"  *)
				m_State:=STATE_CLOSE;
				diError := 16#8003;
			ELSE (* succesful *)
				diError := 16#0000;
				T_Connect(IN:=FALSE);
				(* Copy received data into receive buffer *)
				FOR i:= 0 TO DINT_TO_INT(m_BytesReceived	)-1 DO
					aReceiveBuffer[diReceiveCount]:= m_ReceiveBuffer[i];
					diReceiveCount:=(diReceiveCount+1) MOD SIZEOF(aReceiveBuffer);
				END_FOR

			END_CASE

	(* -------------------------------------------------------------------------*)
	STATE_CLOSE : (* close socket *)
		IF ADR(%MW0)=16#30000000  OR ADR(%MW0)=16#20000000 THEN (*841 or 881*)
			;
		ELSE
			SysSockShutdown(m_Socket, 0);;(*870*)
		END_IF
		m_xReturn := SysSockClose( m_Socket);
		m_Socket := -1;
		m_State := 0; (* succesful *)
		xConnected:=FALSE;
		T_Connect(IN:=FALSE);
	(* -------------------------------------------------------------------------*)
	STATE_ERROR_TRAP: (* error handling *)
		xConnected:=FALSE;

	ELSE  (* Bad FSM code trap  *)
			m_State:= STATE_ERROR_TRAP;
			diError:= 16#8008;
	END_CASE

ELSE(*close connection*)
	IF m_Socket >= 0 THEN
		IF ADR(%MW0)=16#30000000  OR ADR(%MW0)=16#20000000 THEN (*841 or 881*)
			;
		ELSE
			SysSockShutdown(m_Socket, 0);;(*870*)
		END_IF
		SysSockClose( m_Socket);
	END_IF
	m_Socket := -1;
	diError := 16#0000;
	m_State := STATE_CREATE;
	xConnected:=FALSE;
	T_Connect(IN:=FALSE);
END_IF
END_FUNCTION_BLOCK

(* POU Utils Functions/DWORDSWAP, ST *)
FUNCTION DWORDSWAP:BOOL
VAR_INPUT
	pIn:POINTER TO ARRAY[1..4] OF BYTE;
	pOut:POINTER TO ARRAY[1..4] OF BYTE;
END_VAR
VAR
END_VAR
pOut^[1]:=pIn^[4];
pOut^[2]:=pIn^[3];
pOut^[3]:=pIn^[2];
pOut^[4]:=pIn^[1];
END_FUNCTION

(* POU Utils Functions/CHKSTRING, ST *)
FUNCTION CHKSTRING : BOOL
VAR_INPUT
	pString: POINTER TO BYTE;
	pPattern: POINTER TO BYTE;
END_VAR
VAR
END_VAR
CHKSTRING:=TRUE;
WHILE pPattern^<>0 AND CHKSTRING DO
	IF pPattern^<>pString^ THEN CHKSTRING:=FALSE; END_IF
	pString:=pString+1;
	pPattern:=pPattern+1;
END_WHILE
END_FUNCTION

(* POU TCP_Remote/Remote_Proc, ST *)
PROGRAM Remote_Proc
VAR
	s1:         	TCPSERVER;
	Enable: 		BOOL;
	Connected: 		BOOL;
	Error: 			DINT;

	TxData:			ARRAY [0..MAX_SEND_TCP_SERVER] OF BYTE;
	TxLen:			DINT;
	TxTrig:			BOOL;

	RxData:			ARRAY [0..MAX_RECEIVE_TCP_SERVER] OF BYTE;
	RxLen:			DINT;

	Status:			DINT;

	(* Command interpreter *)

	Cmd_Buf:		ARRAY [0..MAX_RECEIVE_TCP_SERVER] OF BYTE;
	Cmd_Buf_U16:	POINTER TO WORD;
	Cmd_Buf_INT:	POINTER TO INT;
	Cmd_BufLen:		WORD;
	Cmd_St:			WORD;

	Cmd_Obj:		WORD;
	Cmd_ObjIdx:		WORD;
	Cmd_C:			WORD;
	Cmd_R:			WORD;
	Cmd_CLen:		WORD;
	Cmd_RLen:		WORD;

	i : WORD;
	j : INT;
	s2 : STRING;

END_VAR
(*=== State machine ===*)
CASE Status OF
	0: (* Startup *)
		TxLen:=0; TxTrig:=FALSE;
		RxLen:=0;
		Enable:=TRUE;
		Status:=1;

	1: (* Wait incoming connection *)
		IF Connected THEN
			(* Log access *)(*
			LogEv(EL_Log,EO_VPN,1,5,'Remote');*)
			(* Send welcome message *)(*
			ADDSTRING(pTxData:=ADR(TxData), pString:=ADR(Remote_WELCOME), TxLen:=TxLen);
			TxTrig:=TRUE;*)
			(* Reset vars *)
			Cmd_BufLen:=0;
			Cmd_St:=0;
			Status:=2;
		END_IF
		IF Error>1 THEN
			Enable:=FALSE;
			Status:=0;
		END_IF

	2: (* Wait command *)
		IF RxLen>0 THEN
			(*=== Interpreter start ===*)
			IF Cmd_BufLen+(RxLen/2)>=MAX_RECEIVE_TCP_SERVER THEN
				(* ERROR *)
				Cmd_BufLen:=0;
			ELSE
				i:=HEXTORAW(pString:=ADR(RxData), StringLen:=DINT_TO_WORD(RxLen), pData:=ADR(Cmd_Buf[Cmd_BufLen]));
				Cmd_BufLen:=Cmd_BufLen+i;
			END_IF
			IF Cmd_BufLen>=8 THEN
				Cmd_Buf_U16:=ADR(Cmd_Buf[6]);
				IF Cmd_BufLen>=(8+Cmd_Buf_U16^) THEN
					Cmd_CLen:=Cmd_Buf_U16^;
					Cmd_Buf_U16:=ADR(Cmd_Buf[0]); Cmd_Obj:=Cmd_Buf_U16^;
					Cmd_Buf_U16:=ADR(Cmd_Buf[2]); Cmd_ObjIdx:=Cmd_Buf_U16^;
					Cmd_Buf_U16:=ADR(Cmd_Buf[4]); Cmd_C:=Cmd_Buf_U16^;
					(* Log command *)(*
					s2:='RCmd_';		s2:=CONCAT(s2,WORD_TO_STRING(Cmd_Obj));
					s2:=CONCAT(s2,'_'); s2:=CONCAT(s2,WORD_TO_STRING(Cmd_ObjIdx));
					s2:=CONCAT(s2,'_'); s2:=CONCAT(s2,WORD_TO_STRING(Cmd_C));
					s2:=CONCAT(s2,'_');	s2:=CONCAT(s2,WORD_TO_STRING(Cmd_CLen));
					LogEv(EL_Log,EO_VPN,1,6,s2);*)
					(* Execute command *)
					Command();
					Cmd_BufLen:=0;
				END_IF
			END_IF
			(*=== Interpreter end ===*)
			RxLen:=0;
		END_IF
		IF NOT Connected THEN
			Status:=0;
		END_IF

ELSE
	Status:=0;
END_CASE


(*=== Execute server lib ===*)
s1(
	xEnable				:= Enable,
	wPortNumber			:= Remote_PORT,
	tServerTimeOut		:= t#15m,
	ptSendData			:= ADR(TxData),
	diSendCount			:= TxLen,
	xStartSend			:= TxTrig,
	aReceiveBuffer		:= RxData,
	diReceiveCount		:= RxLen,
	xClientConnected	=> Connected,
	diError				=> Error
);
END_PROGRAM
ACTION Cmd_CAL:
(* Check index *)(*
IF Cmd_ObjIdx<1 OR Cmd_ObjIdx>2 THEN
	Cmd_R:=2;
	RETURN;
END_IF

(* Process command *)
CASE Cmd_C OF

	3: (* TRY REARM *)
		IF Cmd_ObjIdx=1 THEN
			CAL01.Rearm:=TRUE;
		ELSE
			CAL02.Rearm:=TRUE;
		END_IF

ELSE
	Cmd_R:=3;
END_CASE
*);
END_ACTION
ACTION Cmd_CRON:
(* Check index *)
IF Cmd_ObjIdx<1 OR Cmd_ObjIdx>6 THEN
	Cmd_R:=2;
	RETURN;
END_IF

(* Process command *)
CASE Cmd_C OF

	1: (* GET PROFILE *)
		IF Cmd_CLen<>3 THEN
			Cmd_R:=4;
		ELSE
			(* Load profile *)
			CronEd.CN_Sel:=WORD_TO_BYTE(Cmd_ObjIdx);
			Cmd_Buf_U16:=ADR(Cmd_Buf[8]);
			CronEd.CN_YSel:=Cmd_Buf_U16^;
			CronEd.PR_Sel:=Cmd_Buf[10];
			CronEd.PR_Load_Exe();
			(* Copy data *)
			Cmd_RLen:=192;
			TxLen:=TxLen+RAWTOHEX(ADR(CronEd.PR.Setpoint),192,ADR(TxData[TxLen]));
		END_IF

	2: (* SET PROFILE *)
		IF Cmd_CLen<>(3+192) THEN
			Cmd_R:=4;
		ELSE
			(* Save profile *)
			CronEd.CN_Sel:=WORD_TO_BYTE(Cmd_ObjIdx);
			Cmd_Buf_U16:=ADR(Cmd_Buf[8]);
			CronEd.CN_YSel:=Cmd_Buf_U16^;
			CronEd.PR_Sel:=Cmd_Buf[10];
			MEMCPY(ADR(Cmd_Buf[11]),ADR(CronEd.PR.Setpoint),192);
			CronEd.PR_Save_Exe();
		END_IF

	5: (* GET CALENDAR MONTH *)
		IF Cmd_CLen<>3 THEN
			Cmd_R:=4;
		ELSE
			(* Load calendar *)
			CronEd.CN_Sel:=WORD_TO_BYTE(Cmd_ObjIdx);
			Cmd_Buf_U16:=ADR(Cmd_Buf[8]);
			CronEd.CN_YSel:=Cmd_Buf_U16^;
			CronEd.CA_Sel:=Cmd_Buf[10];
			CronEd.CA_Load_Exe();
			(* Copy data *)
			Cmd_RLen:=32;
			TxLen:=TxLen+RAWTOHEX(ADR(CronEd.CA.Profile),32,ADR(TxData[TxLen]));
		END_IF

	6: (* SET CALENDAR MONTH *)
		IF Cmd_CLen<>(3+32) THEN
			Cmd_R:=4;
		ELSE
			(* Save calendar *)
			CronEd.CN_Sel:=WORD_TO_BYTE(Cmd_ObjIdx);
			Cmd_Buf_U16:=ADR(Cmd_Buf[8]);
			CronEd.CN_YSel:=Cmd_Buf_U16^;
			CronEd.CA_Sel:=Cmd_Buf[10];
			MEMCPY(ADR(Cmd_Buf[11]),ADR(CronEd.CA.Profile),32);
			CronEd.CA_Save_Exe();
		END_IF

	9: (* CRON RESTART *)
		CASE Cmd_ObjIdx OF
			1: CRON01.InitOK:=FALSE;
			2: CRON02.InitOK:=FALSE;
			3: CRON03.InitOK:=FALSE;
			4: CRON04.InitOK:=FALSE;
			5: CRON05.InitOK:=FALSE;
			6: CRON06.InitOK:=FALSE;
			7: CRON07.InitOK:=FALSE;
			8: CRON08.InitOK:=FALSE;
			9: CRON09.InitOK:=FALSE;
			10: CRON10.InitOK:=FALSE;
			11: CRON11.InitOK:=FALSE;
			12: CRON12.InitOK:=FALSE;
			13: CRON13.InitOK:=FALSE;
			14: CRON14.InitOK:=FALSE;
		END_CASE

ELSE
	Cmd_R:=3;
END_CASE
END_ACTION
ACTION Cmd_LUX:
(* Check index *)
IF Cmd_ObjIdx<1 OR Cmd_ObjIdx>6 THEN
	Cmd_R:=2;
	RETURN;
END_IF


(* Process command *)
CASE Cmd_C OF

	0:	(* Restore default functioning mode *)
		CASE Cmd_ObjIdx OF

			1:	LUX01.RestoreMode(WORKINGTIME:=LuxWT[1], POWERONCYCLES:=LuxPOC[1]);
			2:	LUX02.RestoreMode(WORKINGTIME:=LuxWT[2], POWERONCYCLES:=LuxPOC[2]);
			3:	LUX03.RestoreMode(WORKINGTIME:=LuxWT[3], POWERONCYCLES:=LuxPOC[3]);
			4:	LUX04.RestoreMode(WORKINGTIME:=LuxWT[4], POWERONCYCLES:=LuxPOC[4]);
			5:	LUX05.RestoreMode(WORKINGTIME:=LuxWT[5], POWERONCYCLES:=LuxPOC[5]);
			6:	LUX06.RestoreMode(WORKINGTIME:=LuxWT[6], POWERONCYCLES:=LuxPOC[6]);

		END_CASE

	1:	(* Reset statistic counter *)
		CASE Cmd_ObjIdx OF

			1:	LUX01.StatReset(WORKINGTIME:=LuxWT[1], POWERONCYCLES:=LuxPOC[1]);
			2:	LUX02.StatReset(WORKINGTIME:=LuxWT[2], POWERONCYCLES:=LuxPOC[2]);
			3:	LUX03.StatReset(WORKINGTIME:=LuxWT[3], POWERONCYCLES:=LuxPOC[3]);
			4:	LUX04.StatReset(WORKINGTIME:=LuxWT[4], POWERONCYCLES:=LuxPOC[4]);
			5:	LUX05.StatReset(WORKINGTIME:=LuxWT[5], POWERONCYCLES:=LuxPOC[5]);
			6:	LUX06.StatReset(WORKINGTIME:=LuxWT[6], POWERONCYCLES:=LuxPOC[6]);

		END_CASE

ELSE
	Cmd_R:=3;
END_CASE
END_ACTION
ACTION Cmd_SYS:
(* Check index *)
IF Cmd_ObjIdx<>0 THEN
	Cmd_R:=2;
	RETURN;
END_IF

(* Process command *)
CASE Cmd_C OF

	0: (* ECHO *)
		IF Cmd_CLen<>0 THEN
			TxLen:=0;
		END_IF

	1: (* LOG REQUEST *)
		LogTrig();

	2: (* REARM *)
		Sys.Warning:=FALSE;
		Sys.Alarm:=FALSE;
		Sys.AlarmStop:=FALSE;

	3: (* GET INFO1 *)
		Cmd_RLen:=6;
		TxLen:=TxLen+RAWTOHEX(ADR(Plant_SN),4,ADR(TxData[TxLen]));
		TxLen:=TxLen+RAWTOHEX(ADR(Plant_SW_VER),2,ADR(TxData[TxLen]));

ELSE
	Cmd_R:=3;
END_CASE
END_ACTION
ACTION Command:
(* Default response OK/NODATA *)
Cmd_R:=0;
Cmd_RLen:=0;
TxLen:=16;

(* Check object *)
CASE Cmd_Obj OF

	EO_SYS:
		Cmd_SYS();

	EO_CRON:
		Cmd_CRON();

	EO_LUX:
		Cmd_LUX();

ELSE
	Cmd_R:=3;
END_CASE

(* Generate response *)
IF TxLen>0 THEN
	RAWTOHEX(ADR(Cmd_Obj)	,2,ADR(TxData[ 0]));
	RAWTOHEX(ADR(Cmd_ObjIdx),2,ADR(TxData[ 4]));
	RAWTOHEX(ADR(Cmd_R)		,2,ADR(TxData[ 8]));
	RAWTOHEX(ADR(Cmd_RLen)	,2,ADR(TxData[12]));
	TxTrig:=TRUE;
END_IF
END_ACTION

(* POU Utils Functions/TCPSERVER, ST *)
FUNCTION_BLOCK TCPSERVER
(***********************************************************************************************************	*)
(* Version: 1.6                                    			          											*)
(* Date: 11.02.2011                                   					          							    *)
(***********************************************************************************************************	*)
(* WAGO Kontakttechnik GmbH Hansastr. 27 32423 Minden(Westf.)													*)
(* Tel. +0049 571/887-0 Fax. +0049 571/887-0																	*)
(* Author: VB																									*)
(***********************************************************************************************************	*)
(*Description:	A TCP server to read and write data													       		*)
(*Historie:																										*)
(*Version 1.6: 11.02.2011: Changes according to 750-880/881											 			*)
(*Version 1.5: 27.11.2008 Bugfix allow reuse port																*)
(*Version 1.4: 13.10.2008 Bugfix transmitting large data														*)
(*Version 1.3: 15.01.2007 Changes according to FW11																*)
(*Version 1.2: 09.03.2006 Changes for socket handle 0											       			*)
(*Version 1.1: 14.02.2005 Release																				*)
(***********************************************************************************************************	*)
VAR CONSTANT
	STATE_INIT     				 : BYTE:= 0;
	STATE_OPEN     				 : BYTE:= 1;
	STATE_TX       				 : BYTE:= 20;
	STATE_RX       				 : BYTE:= 30;
	STATE_CLOSE    				 : BYTE:= 40;
	STATE_ERROR_TRAP		 	 : BYTE:= 200;
END_VAR
VAR_INPUT
	xEnable    					: BOOL;	 (* Set TRUE to enable function block *)
	wPortNumber					: WORD;  (* Port *)
	tServerTimeOut				: TIME:=t#50s;
	ptSendData					: POINTER TO ARRAY[0..MAX_SEND_TCP_SERVER] OF BYTE;
	diSendCount					: DINT;
END_VAR
VAR_OUTPUT
	xClientConnected  			: BOOL:= FALSE;
	diError 					: DINT:= 0;
END_VAR
(* Status Codes -----------------------------------------
	16#8001 => No socket descriptor available 
	16#8002 => SysSockBind fails 
	16#8003 => SysSockListen fails 
	16#8004 => switching to none blocking mode fails
	16#8005 => SysSockClose() returns FALSE 
    16#8006 => SysSockConnect() fails
    16#8007 => SysSockSend() fails
	16#8008 => error state machine 
	16#8009 => timeout while waiting for data from server 
	16#0001 => server waiting for client to establish connection
------------------------------------------------------------*)
VAR_IN_OUT
	xStartSend					: BOOL;
	aReceiveBuffer				: ARRAY [0..MAX_RECEIVE_TCP_SERVER] OF BYTE;
	diReceiveCount				: DINT;
END_VAR

VAR
	m_State    					: BYTE:= 0;
	m_ReceiveBuffer				: ARRAY [0..MAX_RECEIVE_TCP_SERVER_SOCKET] OF BYTE;
	m_ServerSocket				: DINT:= SOCKET_INVALID;
	m_Socket					: DINT:= SOCKET_INVALID;
	m_AddressInfo				: SOCKADDRESS;
	m_BytesReceived				: DINT;
	m_diReturn					: DINT;
	m_xReturn					: BOOL;
	m_SizeSockadr				: DWORD;
	m_ConnectionWatchdog		: TON;
	m_Flags						: DINT;
	m_NoneBlocking   			: DINT:= 1;
	m_Blocking   				: DINT:= 0;
	i							: INT;
	m_count						: DINT;
	diOption					: DINT := 1;
	on: DINT;
END_VAR
IF xEnable THEN
	CASE m_State OF
		STATE_INIT:
			(* Create Socket *)
			m_ServerSocket:= SysSockCreate( SOCKET_AF_INET, SOCKET_STREAM, 0);
			IF m_ServerSocket = SOCKET_INVALID THEN
				(* *)
				diError:= 16#8001;
				m_State:= STATE_ERROR_TRAP;
				RETURN;
			ELSE
				;
			END_IF
			(* Address bindings *)
			(********************)
			on:=1;
			SysSockSetOption( m_ServerSocket, SOCKET_SOL, SOCKET_SO_REUSEADDR, ADR(on), SIZEOF(on) );

			m_AddressInfo.sin_family:= SOCKET_AF_INET;
			m_AddressInfo.sin_port  := SysSockHtons( wPortNumber);
			m_AddressInfo.sin_addr  := SOCKET_INADDR_ANY;
			IF NOT SysSockBind( m_ServerSocket, ADR(m_AddressInfo), SIZEOF(m_AddressInfo)) THEN
				diError:= 16#8002;
				m_State:= STATE_ERROR_TRAP;
				RETURN;
			END_IF
			(* Wait for connections *)
			(************************)
			IF NOT SysSockListen( m_ServerSocket, 1) THEN
				diError:= 16#8003;
				m_State:= STATE_ERROR_TRAP;
			END_IF

			(* Puts SOCKET in NonBlocking mode *)
			m_diReturn:= SysSockIoctl( m_ServerSocket, SOCKET_FIONBIO, ADR(m_NoneBlocking));

			m_State:= STATE_OPEN;


		STATE_OPEN: 	(* Waiting for incomming connection *)
				m_SizeSockadr:=SIZEOF(m_AddressInfo);
				m_Socket:= SysSockAccept( m_ServerSocket, ADR(m_AddressInfo), ADR(m_SizeSockadr));
				diError:=State_open;
				IF m_Socket <> SOCKET_INVALID THEN
					xClientConnected:=TRUE;
					(*Set Push-Bit:new V1.5*)
					IF ADR(%MW0)=16#30000000  OR ADR(%MW0)=16#20000000 THEN (*841 or 881*)
						SysSockSetOption(
							diSocket:=m_Socket,
							diLevel:=6,
							diOption:=SOCKET_TCP_NODELAY,
							pOptionValue:=ADR(diOption),
							diOptionLength:=SIZEOF(diOption));
					ELSE
							;
					END_IF
					SysSockIoctl( m_Socket, SOCKET_FIONBIO, ADR(m_NoneBlocking));
					m_State:= STATE_RX;
					diError:=0;
				END_IF

		STATE_RX:
					m_BytesReceived:= SysSockRecv( m_Socket, ADR(m_ReceiveBuffer), SIZEOF(m_ReceiveBuffer), 0);
					CASE m_BytesReceived OF
					-1:(*no data available or error occured*)
						m_ConnectionWatchdog(IN:=TRUE , PT:=tServerTimeOut );
						IF m_connectionWatchdog.Q THEN
							m_State:= STATE_CLOSE;
							m_ConnectionWatchdog(IN:=FALSE);(*reset connection watchdog*)
							diError := 16#8009;
						END_IF
					0:(* socket was "gracefully closed"  *)
						m_State:= STATE_CLOSE;
						diError := 16#8003;
					ELSE
						(* Copy received data into receive buffer *)
						(********************************)
						FOR i:= 0 TO DINT_TO_INT(m_BytesReceived	)-1 DO
							aReceiveBuffer[diReceiveCount]:= m_ReceiveBuffer[i];
							diReceiveCount:=(diReceiveCount+1) MOD SIZEOF(aReceiveBuffer);
						END_FOR

						m_ConnectionWatchdog(IN:=FALSE);(*reset connection watchdog*)
					END_CASE

				(*send data*)
				IF xStartSend	 THEN
					m_State := STATE_TX;
				END_IF

	STATE_TX:	 (* send TCP-message *)
		m_diReturn := SysSockSend(diSocket := m_Socket,
								  pbyBuffer := ADR(ptSendData^[m_count]),(*geändert V1.4 bisher: [0] *)
								  diBufferSize := diSendCount-m_count,
								  diFlags :=m_Flags);
		CASE m_diReturn OF
		-1:	(* ERROR or data could not yet be send (V1.3 due to new FW11) *)
			m_ConnectionWatchdog(IN:=TRUE , PT:=tServerTimeOut );
			IF m_connectionWatchdog.Q THEN
				m_State:= STATE_CLOSE;
				m_ConnectionWatchdog(IN:=FALSE);(*reset connection watchdog*)
				diError := 16#8007;
			END_IF
		0: (* socket was "gracefully closed"  *)
			m_State := STATE_CLOSE;
			diError := 16#8003;
		ELSE (* succesful *)
			m_count:=m_count+m_diReturn;
			IF m_count>=diSendCount THEN
				diError := 16#0000;
				m_State := STATE_RX;
				m_count:=0;
				xStartSend:=FALSE;
			END_IF
			m_ConnectionWatchdog(IN:=FALSE);(*reset connection watchdog*)
		END_CASE


		STATE_CLOSE:	(* Close the server *)

		IF ADR(%MW0)=16#30000000  OR ADR(%MW0)=16#20000000 THEN (*841 or 881*)
			;
		ELSE
			IF m_Socket>=0 THEN
				SysSockShutdown(m_Socket, 0);;(*870*)
			END_IF
		END_IF
		IF m_Socket>=0 THEN
			SysSockClose( m_Socket);
		END_IF
		xClientConnected:= FALSE;
		m_State:= STATE_OPEN; (* Try to open the server again *)
		m_ConnectionWatchdog(IN:=FALSE);(*reset connection watchdog*)

		STATE_ERROR_TRAP: (* Error Read/Write socket  *)
			m_State:= STATE_ERROR_TRAP;

	ELSE  (* Bad FSM code trap  *)
			m_State:= STATE_ERROR_TRAP;
			diError:= 16#8008;
	END_CASE;
ELSE
	IF m_State <> STATE_INIT THEN
		IF ADR(%MW0)=16#30000000  OR ADR(%MW0)=16#20000000 THEN (*841 or 881*)
			;
		ELSE
			IF m_Socket>=0 THEN
				SysSockShutdown(m_Socket, 0);;(*870*)
			END_IF
		END_IF
		IF m_Socket>=0 THEN
			SysSockClose( m_Socket);
		END_IF
		IF ADR(%MW0)=16#30000000  OR ADR(%MW0)=16#20000000 THEN (*841 or 881*)
			;
		ELSE
			IF m_ServerSocket>=0 THEN
				SysSockShutdown(m_ServerSocket, 0);;(*870*)
			END_IF
		END_IF
		IF m_ServerSocket>=0 THEN
			SysSockClose( m_ServerSocket);
		END_IF
		xClientConnected:= FALSE;
		diError:= 0;
		m_State:= STATE_init; (* Try to open the server again *)
		m_ConnectionWatchdog(IN:=FALSE);(*reset connection watchdog*)
	END_IF
END_IF
END_FUNCTION_BLOCK

(* POU Utils Functions/HEXTORAW, ST *)
FUNCTION HEXTORAW : WORD
VAR_INPUT
	pString		: POINTER TO BYTE;
	StringLen	: WORD;
	pData		: POINTER TO BYTE;
END_VAR
VAR
	xl: WORD;
	xi: WORD;
	xr: BYTE;
END_VAR
xl:=0;
xi:=0;

WHILE xi<StringLen DO

	IF pString^>=97 AND pString^<=102 THEN
		xr := pString^ - 87;
	ELSIF pString^>=65 AND pString^<=70 THEN
		xr := pString^ - 55;
	ELSIF pString^>=48 AND pString^<=57 THEN
		xr := pString^ - 48;
	ELSE
		xr := 16;
	END_IF

	IF xr<16 THEN
		IF (xi AND 1)=0 THEN
			pData^ := xr * 16;
		ELSE
			pData^ := pData^ + xr;
			pData := pData + 1;
			xl := xl + 1;
		END_IF
	END_IF

	xi := xi + 1;
	pString := pString + 1;

END_WHILE

HEXTORAW:=xl;
END_FUNCTION

(* POU Utils Functions/RAWTOHEX, ST *)
FUNCTION RAWTOHEX : WORD
VAR_INPUT
	pData: POINTER TO BYTE;
	DataLen: WORD;
	pString: POINTER TO BYTE;
END_VAR
VAR
	xl: WORD;
END_VAR
xl:=0;

WHILE DataLen>0 DO

	pString^ := (pData^ / 16#10) + 48 + (((pData^ / 16#10)/10)*7);
	pString:=pString+1;
	pString^ := (pData^ AND 16#0F)  + 48 + (((pData^ AND 16#0F)/10)*7);
	pString:=pString+1;
	pData:=pData+1;
	DataLen:=DataLen-1;
	xl:=xl+2;

END_WHILE

(*pString^:=0;*)

RAWTOHEX:=xl;
END_FUNCTION

(* POU Utils/USRLED_Update, ST *)
PROGRAM USRLED_Update
VAR
	OldStatus: en_SYS_Status;

	aFS : ARRAY [0..24] OF FLASHING_SEQUENCE :=
		(Colour:=GREEN,  Frequency:=1,   Relation:=128, Duration:=t#0s,    NextIndex:=0),  (* 0 => RUNNING *)
		(Colour:=ORANGE, Frequency:=1,   Relation:=128, Duration:=t#0s,    NextIndex:=1),  (* 1 => INIT *)
		(Colour:=RED,    Frequency:=4,   Relation:=128, Duration:=t#0s,    NextIndex:=2),  (* 2 => ERROR *)
		(Colour:=RED,    Frequency:=10,  Relation:=128, Duration:=t#0s,    NextIndex:=3),  (* 3 => ALARM *)
		(Colour:=ORANGE, Frequency:=200, Relation:=16,  Duration:=t#100ms, NextIndex:=11), (* 10 *)
		(Colour:=ORANGE, Frequency:=200, Relation:=32,  Duration:=t#100ms, NextIndex:=12),
		(Colour:=ORANGE, Frequency:=200, Relation:=64,  Duration:=t#100ms, NextIndex:=13),
		(Colour:=ORANGE, Frequency:=200, Relation:=128, Duration:=t#100ms, NextIndex:=14),
		(Colour:=ORANGE, Frequency:=200, Relation:=192, Duration:=t#100ms, NextIndex:=15),
		(Colour:=ORANGE, Frequency:=200, Relation:=128, Duration:=t#100ms, NextIndex:=16),
		(Colour:=ORANGE, Frequency:=200, Relation:=64,  Duration:=t#100ms, NextIndex:=17),
		(Colour:=ORANGE, Frequency:=200, Relation:=32,  Duration:=t#100ms, NextIndex:=18),
		(Colour:=ORANGE, Frequency:=200, Relation:=16,  Duration:=t#100ms, NextIndex:=19),
		(Colour:=ORANGE, Frequency:=200, Relation:=8,   Duration:=t#100ms, NextIndex:=10),
		(Colour:=GREEN,  Frequency:=200, Relation:=16,  Duration:=t#100ms, NextIndex:=21), (* 20 *)
		(Colour:=GREEN,  Frequency:=200, Relation:=32,  Duration:=t#100ms, NextIndex:=22),
		(Colour:=GREEN,  Frequency:=200, Relation:=64,  Duration:=t#100ms, NextIndex:=23),
		(Colour:=GREEN,  Frequency:=200, Relation:=128, Duration:=t#100ms, NextIndex:=24),
		(Colour:=GREEN,  Frequency:=200, Relation:=192, Duration:=t#100ms, NextIndex:=25),
		(Colour:=GREEN,  Frequency:=200, Relation:=128, Duration:=t#100ms, NextIndex:=26),
		(Colour:=GREEN,  Frequency:=200, Relation:=64,  Duration:=t#100ms, NextIndex:=27),
		(Colour:=GREEN,  Frequency:=200, Relation:=32,  Duration:=t#100ms, NextIndex:=28),
		(Colour:=GREEN,  Frequency:=200, Relation:=16,  Duration:=t#100ms, NextIndex:=29),
		(Colour:=GREEN,  Frequency:=200, Relation:=8,   Duration:=t#100ms, NextIndex:=20);

	pFS : POINTER TO FLASHING_SEQUENCE;


END_VAR
IF Sys.Status <> OldStatus THEN

	OldStatus:=Sys.Status;

	CASE OldStatus OF

		S_STARTUP:
			pFS:=ADR(aFS);
			SET_FLASHING_SEQUENCE(EN:=TRUE, POINTER_TO_POINTER_TO_ARRAY:=ADR(pFS));
			SET_FLASHING_SEQUENCE_INDEX(EN:=TRUE, IMMEDIATE:=FALSE, INDEX:=1);
			START_FLASHING_SEQUENCE(EN:=TRUE);

		S_RUNNING:
			SET_FLASHING_SEQUENCE_INDEX(EN:=TRUE, IMMEDIATE:=TRUE, INDEX:=0);

	END_CASE

END_IF
END_PROGRAM

(* POU Configuration/MODBUS_CONFIGURATION, ST *)
PROGRAM MODBUS_CONFIGURATION        
VAR                                
END_VAR                            
(*                                 
   <?xml version="1.0" encoding="UTF-16" standalone="yes"?>
<network xml_structure_version="1">
	<generator_settings minRTUTaskCycleTimeMs="5" minEthaskCycleTimeMs="5" ethSlaveMultiplier="0.1" rtuInterfaceMultiplier="0.1" taskGeneration="false"/>
</network>
                              
*)                                 
;                                  
END_PROGRAM

(* POU Plant/SCA_Proc, ST *)
PROGRAM SCA_Proc
VAR
	SCA01_1	:	FLT_TAP;
	SCA01_2	:	FLT_TAP;
	SCA01_3	:	FLT_TAP;

	upd		:	BOOL;
END_VAR
(***** SCA01 *****)
SCA01_1(IN:=SCA01_1_DI);
IF SCA01_1.EVL THEN LogEv(EL_Wrn,EO_SCA,1,1,'1'); upd:=TRUE; END_IF
IF SCA01_1.EVH THEN	LogEv(EL_Log,EO_SCA,1,2,'1'); upd:=TRUE; END_IF

SCA01_2(IN:=SCA01_2_DI);
IF SCA01_2.EVL THEN	LogEv(EL_Wrn,EO_SCA,1,1,'2'); upd:=TRUE; END_IF
IF SCA01_2.EVH THEN	LogEv(EL_Log,EO_SCA,1,2,'2'); upd:=TRUE; END_IF

SCA01_3(IN:=SCA01_3_DI);
IF SCA01_3.EVL THEN	LogEv(EL_Wrn,EO_SCA,1,1,'3'); upd:=TRUE; END_IF
IF SCA01_3.EVH THEN	LogEv(EL_Log,EO_SCA,1,2,'3'); upd:=TRUE; END_IF

IF upd THEN
	upd:=FALSE;
	Logger_Head();
	AddLogData();
	Logger_Send();
END_IF
END_PROGRAM
ACTION AddLogData:
Logger.s1:='&SCA01=';
Logger.s1:=CONCAT(Logger.s1,BYTE_TO_STRING(BOOL_TO_BYTE(SCA01_1.OUT))		); Logger.s1:=CONCAT(Logger.s1,';');
Logger.s1:=CONCAT(Logger.s1,BYTE_TO_STRING(BOOL_TO_BYTE(SCA01_2.OUT))		); Logger.s1:=CONCAT(Logger.s1,';');
Logger.s1:=CONCAT(Logger.s1,BYTE_TO_STRING(BOOL_TO_BYTE(SCA01_3.OUT))		);
ADDSTRING(ADR(Logger.TData), ADR(Logger.s1), Logger.TLen);
END_ACTION

(* POU Utils Functions/FLT_TAP, ST *)
FUNCTION_BLOCK FLT_TAP
VAR_INPUT
	IN		: BOOL;
	TAP		: BYTE:=4;
	INITEV	: BOOL:=TRUE;
END_VAR
VAR_OUTPUT
	OUT		: BOOL;
	EVH		: BOOL;
	EVL		: BOOL;
END_VAR
VAR
	init	: BOOL:=FALSE;
	cnt		: BYTE;
END_VAR
EVH:=FALSE;
EVL:=FALSE;

IF NOT init THEN
	init := TRUE;
	IF INITEV THEN
		OUT  := NOT IN;
		cnt  := TAP;
	ELSE
		OUT  := IN;
	END_IF
END_IF

IF OUT<>IN THEN
	cnt:=cnt+1;
	IF cnt>TAP THEN
		OUT:=IN;
		cnt:=0;
		IF OUT THEN EVH:=TRUE; ELSE EVL:=TRUE; END_IF
	END_IF
ELSE
	cnt:=0;
END_IF
END_FUNCTION_BLOCK

(* POU TCP_Logger/LogEv, ST *)
FUNCTION LogEv : BOOL
VAR_INPUT
	Level	: en_Logger_ErrLev;
	Object  : en_SYS_Objects;
	Index	: WORD;
	Error	: WORD;
	Message : STRING;
END_VAR
VAR
	s1 : STRING(160);
	i  : INT;
END_VAR
(* Execute error level operations *)
CASE Level OF
	EL_Wrn: 		Sys.Warning:=TRUE;
	EL_Alarm: 		Sys.Alarm  :=TRUE;
	EL_AlarmStop: 	Sys.Alarm  :=TRUE; (* GO TO STOP STATE!! *)
END_CASE

(* Fill lastlog list *)
s1:=CONCAT(Sys.Time_LogString,';Lev=');
s1:=CONCAT(s1,INT_TO_STRING(Level));
s1:=CONCAT(s1,';Obj=');
s1:=CONCAT(s1,INT_TO_STRING(Object));
s1:=CONCAT(s1,';Idx=');
s1:=CONCAT(s1,WORD_TO_STRING(Index));
s1:=CONCAT(s1,';Err=');
s1:=CONCAT(s1,WORD_TO_STRING(Error));
Sys.LastLogs_Dat[Sys.LastLogs_Idx]:=s1;
Sys.LastLogs_Msg[Sys.LastLogs_Idx]:=Message;
Sys.LastLogs_Idx:=Sys.LastLogs_Idx+1;
IF Sys.LastLogs_Idx>5 THEN Sys.LastLogs_Idx:=0; END_IF

(*---------------------------------------------------------------*)
	Logger_Head();
(*---------------------------------------------------------------*)

(* Insert ERR *)
s1:=CONCAT('&ERR=',INT_TO_STRING(Level));
s1:=CONCAT(s1,';');
s1:=CONCAT(s1,INT_TO_STRING(Object));
s1:=CONCAT(s1,';');
s1:=CONCAT(s1,WORD_TO_STRING(Index));
s1:=CONCAT(s1,';');
s1:=CONCAT(s1,WORD_TO_STRING(Error));
s1:=CONCAT(s1,';');
ADDSTRING(ADR(Logger.TData), ADR(s1), Logger.TLen);
s1:=Message;
STR_NOSPACES(ADR(s1));
ADDSTRING(ADR(Logger.TData), ADR(s1), Logger.TLen);

(*---------------------------------------------------------------*)
	Logger_Send();
(*---------------------------------------------------------------*)
END_FUNCTION

(* POU TCP_Logger/Logger_Head, ST *)
FUNCTION Logger_Head : BOOL
VAR
	s1 : STRING(160);
	i  : BYTE;
END_VAR
Logger.TLen:=0;
(* Set GET header *)
ADDSTRING(ADR(Logger.TData), ADR(Logger_GETSTART), Logger.TLen);

(* Insert Header *)
s1:=INSERT('ID=&V=1&D=',DWORD_TO_STRING(Plant_SN),3);
s1:=CONCAT(s1,Sys.Time_LogString);
s1:=CONCAT(s1,'&S=');
IF Sys.Alarm THEN i:=2; ELSIF Sys.Warning THEN i:=1; ELSE i:=0; END_IF
s1:=CONCAT(s1,BYTE_TO_STRING(i));
ADDSTRING(ADR(Logger.TData), ADR(s1), Logger.TLen);
END_FUNCTION

(* POU Utils Functions/ADDSTRING, ST *)
FUNCTION ADDSTRING : BOOL (* Append string to a byte buffer *)
VAR_INPUT
	pTxData: POINTER TO BYTE;
	pString: POINTER TO BYTE;
END_VAR
VAR_IN_OUT
	TxLen: DINT;
END_VAR
VAR
END_VAR
pTxData:=pTxData+TxLen;
WHILE pString^<>0 DO
	pTxData^:=pString^;
	pString:=pString+1;
	pTxData:=pTxData+1;
	TxLen:=TxLen+1;
END_WHILE
END_FUNCTION

(* POU Utils Functions/STR_NOSPACES, ST *)
FUNCTION STR_NOSPACES : BOOL (* Replace spaces and bad chars with allowed ones, used as HTTP-GET validator *)
VAR_INPUT
	pString: POINTER TO BYTE;
END_VAR
VAR
END_VAR
WHILE pString^<>0 DO
	IF pString^=16#20 (* space *) THEN pString^:=16#5F; (*'_'*) END_IF
	pString:=pString+1;
END_WHILE
END_FUNCTION

(* POU TCP_Logger/Logger_Send, ST *)
FUNCTION Logger_Send : BOOL
VAR
	hFile: 	DWORD;
	pos:	DWORD;
END_VAR
(* Finalize string *)
ADDSTRING(ADR(Logger.TData), ADR(Logger_GETEND), Logger.TLen);

(* Read log position *)
pos:=SysFileGetSize(Logger_DataFile);
(* Check log size, bckup and erase if no pending messages *)
IF pos>5000000(*5M*) THEN
	hFile:=SysFileOpen(Logger_IndexFile,'r');
	IF hFile=0 THEN
		SysFileDelete(Logger_DataFileOld);
		SysFileRename(Logger_DataFile,Logger_DataFileOld);
		pos:=0;
	ELSE
		SysFileClose(hFile);
	END_IF
END_IF
(* Write message on log file *)
hFile:=SysFileOpen(Logger_DataFile,'a');
IF hFile<>0 THEN
	SysFileWrite(hFile, ADR(Logger.TData), Logger.TLen);
	SysFileClose(hFile);
ELSE
	Sys.Warning:=TRUE;
END_IF


(* Check logger status *)
IF Logger.SendReq=FALSE THEN
	(* Set log position for recovery *)
	Logger.SendIdx:=pos;
	(* Copy message data *)
	MEMCPY(ADR(Logger.TData),ADR(Logger.SendData),DINT_TO_WORD(Logger.TLen));
	Logger.SendLen:=Logger.TLen;
	(* Trigger request *)
	Logger.SendReq:=TRUE;
ELSE
	(* Add message position+size in recovery indexes *)
	hFile:=SysFileOpen(Logger_IndexFile,'a');
	SysFileWrite(hFile, ADR(pos), SIZEOF(pos));
	SysFileWrite(hFile, ADR(Logger.TLen), SIZEOF(Logger.TLen));
	SysFileClose(hFile);
END_IF
END_FUNCTION

(* POU Utils Functions/MEMCPY, ST *)
FUNCTION MEMCPY:BOOL
VAR_INPUT
	pSourceAddress:POINTER TO ARRAY[1..2] OF BYTE;
	pDestinationAddress:POINTER TO ARRAY[1..2] OF BYTE;
	BytesToCopy:WORD;
END_VAR
VAR
END_VAR
WHILE (BytesToCopy > 0) DO
	pDestinationAddress^[1]:=pSourceAddress^[1]; (* copy bytes from source to destination *)
	pDestinationAddress:=ADR(pDestinationAddress^[2]); (* increment destination *)
	pSourceAddress:=ADR(pSourceAddress^[2]);(* increment source *)
	BytesToCopy:=BytesToCopy -1; (* decrement number of bytes to copy *)
END_WHILE
END_FUNCTION

(* POU Plant/SYS_Proc, ST *)
PROGRAM SYS_Proc
VAR
(*	fALARM_PB		:FLT_TAP;
	fALARM_TB		:FLT_TAP;
	fALARM_PM		:FLT_TAP; *)

(*	fGZB_ST			:FLT_TAP; (* GATEWAY ZIGBEE *)*)
(*	fVPN_OUT1		:FLT_TAP; (* VPN - CONNECT *)*)
	fVPN_OUT2		:FLT_TAP; (* VPN - STATUS *)
(*	fKEY_CT_ST		:FLT_TAP; (* DOOR01 - Porta primaria *)*)
(*	fKEY_SCT_ST		:FLT_TAP; (* DOOR02 - Porta secondaria *)*)
	fKEY_QE_ST		:FLT_TAP; (* DOOR03 - Quadro Elettrico *)

END_VAR
(*************** ISPESL *****************)
(*
fALARM_PB(IN:=ALARM_PB);
IF fALARM_PB.EVH THEN
	LogEv(EL_AlarmStop,EO_PBV,1,1,'Over_Pressure_Alarm');
END_IF

fALARM_TB(IN:=ALARM_TB);
IF fALARM_TB.EVH THEN
	LogEv(EL_AlarmStop,EO_TBV,1,1,'Over_Temperature_Alarm');
END_IF

fALARM_PM(IN:=ALARM_PM);
IF fALARM_PM.EVH THEN
	LogEv(EL_AlarmStop,EO_PMV,1,1,'Under_Pressure_Alarm');
END_IF
*)
(****************************************)

(*### VPN Connection Check ###*)(*
fVPN_OUT1(IN:=VPN_OUT1);
IF fVPN_OUT1.EVH THEN
	LogEv(EL_Log,EO_VPN,1,1,'CONNECT_ON');
END_IF
IF fVPN_OUT1.EVL THEN
	LogEv(EL_Log,EO_VPN,1,2,'CONNECT_OFF');
END_IF*)

(*### VPN Status Check ###*)
fVPN_OUT2(IN:=VPN_OUT2);
IF fVPN_OUT2.EVH THEN
	LogEv(EL_Log,EO_VPN,1,3,'STATUS_UP');
END_IF
IF fVPN_OUT2.EVL THEN
	LogEv(EL_Wrn,EO_VPN,1,4,'STATUS_DOWN');
END_IF

(*### DOOR01 Status Check ###*)(*
fKEY_CT_ST(IN:=KEY_CT_ST);
IF fKEY_CT_ST.EVH THEN
	LogEv(EL_Log,EO_DOOR,1,2,'Centrale_termica_Close');
END_IF
IF fKEY_CT_ST.EVL THEN
	LogEv(EL_Wrn,EO_DOOR,1,1,'Centrale_termica_Open');
END_IF*)

(*### DOOR02 Status Check ###*)(*
fKEY_SCT_ST(IN:=KEY_SCT_ST);
IF fKEY_SCT_ST.EVH THEN
	LogEv(EL_Log,EO_DOOR,2,2,'Sottocentrale_termica_Close');
END_IF
IF fKEY_SCT_ST.EVL THEN
	LogEv(EL_Wrn,EO_DOOR,2,1,'Sottocentrale_termica_Open');
END_IF*)

(*### DOOR03 Status Check ###*)
fKEY_QE_ST(IN:=KEY_QE_ST);
IF fKEY_QE_ST.EVH THEN
	LogEv(EL_Log,EO_DOOR,3,2,'Quadro_Close');
END_IF
IF fKEY_QE_ST.EVL THEN
	LogEv(EL_Wrn,EO_DOOR,3,1,'Quadro_Open');
END_IF
END_PROGRAM

(* POU Utils Functions/AVERAGE_T, ST *)
FUNCTION_BLOCK AVERAGE_T
VAR_INPUT
	IN: 	INT;
END_VAR
VAR_OUTPUT
	HI:		INT;
	AVG:	INT;
	LOW:	INT;
	ERR:	BOOL;
END_VAR
VAR
	sum:	DINT;
	cnt:	WORD;
END_VAR
IF cnt>=65000 THEN
	ERR:=TRUE;
	Read();
	sum := sum - AVG;
	cnt := cnt + 1;
END_IF

sum := sum + IN;
cnt := cnt + 1;

IF IN<LOW THEN  LOW:=IN; END_IF
IF IN>HI  THEN HI :=IN; END_IF
END_FUNCTION_BLOCK
ACTION Read:
AVG := DINT_TO_INT(sum/cnt);
END_ACTION
ACTION Reset:
HI:=IN;
AVG:=IN;
LOW:=IN;
ERR:=FALSE;

sum:=IN;
cnt:=1;
END_ACTION

(* POU Utils Functions/BUILD_16TO32, ST *)
FUNCTION BUILD_16TO32 : DWORD
VAR_INPUT
		pSource	:	POINTER TO WORD;
END_VAR
VAR
		Data	:	DWORD;
END_VAR
Data := WORD_TO_DWORD(pSource^);
pSource := pSource + 1;
Data := Data + WORD_TO_DWORD(pSource^) * 65536;

BUILD_16TO32 := Data;
END_FUNCTION

(* POU Utils Functions/COPY_32SWAP16, ST *)
FUNCTION COPY_32SWAP16:BOOL
VAR_INPUT
	pSourceAddress		:POINTER TO ARRAY[1..2] OF WORD;
	pDestinationAddress	:POINTER TO ARRAY[1..2] OF WORD;
END_VAR
VAR
END_VAR
pDestinationAddress^[1]:=pSourceAddress^[2];
pDestinationAddress^[2]:=pSourceAddress^[1];
END_FUNCTION

(* POU Utils Functions/FLT_EVENT, ST *)
FUNCTION_BLOCK FLT_EVENT
VAR_INPUT
	IN		: BOOL;
	INITEV	: BOOL:=TRUE;
END_VAR
VAR_OUTPUT
	EVH		: BOOL;
	EVL		: BOOL;
END_VAR
VAR
	init	: BOOL:=FALSE;
	old		: BOOL;
END_VAR
EVH:=FALSE;
EVL:=FALSE;

IF NOT init THEN
	init:=TRUE;
	IF INITEV THEN
		old := NOT IN;
	ELSE
		old := IN;
	END_IF
END_IF

IF old<>IN THEN
	old:=IN;
	IF IN THEN EVH:=TRUE; ELSE EVL:=TRUE; END_IF
END_IF
END_FUNCTION_BLOCK

(* POU Utils Functions/FLT_TIME, ST *)
FUNCTION_BLOCK FLT_TIME
VAR_INPUT
	IN		: BOOL;
	TTAP	: TIME:=T#5s;
	INITEV	: BOOL:=TRUE;
END_VAR
VAR_OUTPUT
	OUT		: BOOL;
	EVH		: BOOL;
	EVL		: BOOL;
END_VAR
VAR
	init	: BOOL:=FALSE;
	timer	: TON;
END_VAR
EVH:=FALSE;
EVL:=FALSE;

IF NOT init THEN
	init := TRUE;
	IF INITEV THEN
		OUT  := NOT IN;
	ELSE
		OUT  := IN;
	END_IF
END_IF

IF OUT<>IN THEN
	timer(IN:=TRUE,PT:=TTAP);
	IF timer.Q THEN
		OUT:=IN;
		timer(IN:=FALSE);
		IF OUT THEN EVH:=TRUE; ELSE EVL:=TRUE; END_IF
	END_IF
ELSE
	timer(IN:=FALSE);
END_IF
END_FUNCTION_BLOCK

(* POU TCP_Logger/LogTrig, ST *)
FUNCTION LogTrig : BOOL
VAR
	s1 : STRING(160);
	i  : BYTE;
END_VAR
(*---------------------------------------------------------------*)
	Logger_Head();
(*---------------------------------------------------------------*)


(* Insert contabilizers  *)
ANZ01.AddLogData( ModBus:=MODB01 );
ANZ02.AddLogData( ModBus:=MODB01 );
HVAC01.AddLogData(ModBus:=MODB02);
HVAC02.AddLogData(ModBus:=MODB02);

LUX01.AddLogData(WORKINGTIME:=LuxWT[1], POWERONCYCLES:=LuxPOC[1]);
LUX02.AddLogData(WORKINGTIME:=LuxWT[2], POWERONCYCLES:=LuxPOC[2]);
LUX03.AddLogData(WORKINGTIME:=LuxWT[3], POWERONCYCLES:=LuxPOC[3]);
LUX04.AddLogData(WORKINGTIME:=LuxWT[4], POWERONCYCLES:=LuxPOC[4]);
LUX05.AddLogData(WORKINGTIME:=LuxWT[5], POWERONCYCLES:=LuxPOC[5]);
LUX06.AddLogData(WORKINGTIME:=LuxWT[6], POWERONCYCLES:=LuxPOC[6]);

ZTHL01.AddLogData(ModBus:=MODB03);
ZTHL02.AddLogData(ModBus:=MODB03);
ZTHL03.AddLogData(ModBus:=MODB03);
ZTHL04.AddLogData(ModBus:=MODB03);

(*---------------------------------------------------------------*)
	Logger_Send();
(*---------------------------------------------------------------*)
END_FUNCTION

(* POU Utils Functions/MEAN_VALUE, ST *)
FUNCTION MEAN_VALUE : WORD
VAR_INPUT
		pArray	:	POINTER TO ARRAY [1..2] OF WORD;
		Length	:	WORD;
END_VAR
VAR
		counter	:	WORD;
		Sum		:	DWORD;
		(*Maximum	:	WORD;
		Minimum	:	WORD;*)
END_VAR
Sum := 0;
(*Maximum := 0;
Minimum := 0;*)

FOR counter:=1 TO Length BY 1 DO
	Sum := Sum + WORD_TO_DWORD(pArray^[counter]);

	(*IF pArray^[counter] > Maximum THEN Maximum := pArray^[counter]; END_IF
	IF pArray^[counter] < Minimum THEN Minimum := pArray^[counter]; END_IF*)

END_FOR

(*Sum := Sum - WORD_TO_DWORD(Maximum) - WORD_TO_DWORD(Minimum);
MEAN_VALUE := DWORD_TO_WORD(Sum/(Length-2));*)

MEAN_VALUE := DWORD_TO_WORD(Sum/Length);
END_FUNCTION

(* POU Utils Functions/MEMCLR, ST *)
FUNCTION MEMCLR:BOOL
VAR_INPUT
	pDestinationAddress:POINTER TO ARRAY[1..2] OF BYTE;
	BytesToClear:WORD;
END_VAR
VAR
END_VAR
WHILE (BytesToClear > 0) DO
	pDestinationAddress^[1]:=0;
	pDestinationAddress:=ADR(pDestinationAddress^[2]); (* increment destination *)
	BytesToClear:=BytesToClear -1; (* decrement number of bytes to copy *)
END_WHILE
END_FUNCTION

(* POU Plant_Objects/obj_ANALOG_IN_DIFF, ST *)
FUNCTION_BLOCK obj_ANALOG_IN_DIFF
VAR CONSTANT
	NORMAL_STATE:	BYTE := 0;
	LEARN_STATE	:	BYTE := 1;

	SWITCH_ON	:	BYTE := 0;
	READINGS	:	BYTE := 1;
	SWITCH_OFF	:	BYTE := 2;

	LSamples	:	BYTE := 200;	(* Learn samples *)
	MSamples	:	BYTE := 10;		(* Measure samples *)
END_VAR
VAR_INPUT
	ID		:	BYTE;
	Lines   :	BYTE;

	In1		:	BOOL;
	In2		:	BOOL;
	In3		:	BOOL;
	In4		:	BOOL;

	AdcValue:	WORD;

END_VAR
VAR_OUTPUT

	Out1	:	BOOL;
	Out2	:	BOOL;
	Out3	:	BOOL;
	Out4	:	BOOL;

	Alarm	:	BOOL;

END_VAR
VAR
	LearnState	:	BYTE;
	Combination	:	BYTE := 1;
	LSamplesCtr	:	BYTE := 1;
	MSamplesCtr	:	BYTE := 1;
	ActiveLines	:	BYTE;
	Status		:	BYTE;

	ReadValue	:	WORD;
	Threshold_L	:	WORD;
	Threshold_H	:	WORD;

	aLearning	:	ARRAY [1..LSamples] OF WORD;
	aReading	:	ARRAY [1..MSamples] OF WORD;

	SampleTMR	:	TON :=(PT:=T#10ms);
END_VAR
IF Status=NORMAL_STATE THEN
	(* Wait state -> Bypass this block *)
	Out1 := In1;
	Out2 := In2;
	Out3 := In3;
	Out4 := In4;
ELSE
	(* Learning state *)
	Learning();
END_IF
END_FUNCTION_BLOCK
ACTION CheckThreshold:
(* Check actual rele status according to significant rele (line considered in this application) *)
IF Lines = 1 THEN
	ActiveLines.0 := In1;
ELSIF Lines = 2 THEN
		ActiveLines.0 := In1;
		ActiveLines.1 := In2;
ELSIF Lines = 3 THEN
		ActiveLines.0 := In1;
		ActiveLines.1 := In2;
		ActiveLines.2 := In3;
ELSIF Lines = 4 THEN
		ActiveLines.0 := In1;
		ActiveLines.1 := In2;
		ActiveLines.2 := In3;
		ActiveLines.3 := In4;
END_IF

(* Choose the right threshold according to current lines state (switch on or off) *)
IF ActiveLines = 0 THEN
	Threshold_L := 0;
	Threshold_H := (Lux_ref[ID,1] * FeedbackTolerance)/100;
ELSE
	Threshold_L := (Lux_ref[ID,ActiveLines] * (100-FeedbackTolerance))/100;		(* Low threshold *)
	Threshold_H := (Lux_ref[ID,ActiveLines] * (100+FeedbackTolerance))/100;		(* High threshold *)
END_IF

(* Check Alarm *)
IF ReadValue > Threshold_L AND ReadValue < Threshold_H THEN
	Alarm := FALSE;
ELSE
	Alarm := TRUE;
END_IF
END_ACTION
ACTION Learning:
(* State machine to learn value for each possible combination of lines *)
CASE LearnState OF

	SWITCH_ON:	(* Force switch on of the line and start sampling timer *)

		CASE Combination OF

			1:
				Out1 := TRUE;

			2:
				Out2 := TRUE;

			3:
				Out1 := TRUE;
				Out2 := TRUE;

			4:
				Out3 := TRUE;

			5:
				Out1 := TRUE;
				Out3 := TRUE;

			6:
				Out2 := TRUE;
				Out3 := TRUE;

			7:
				Out1 := TRUE;
				Out2 := TRUE;
				Out3 := TRUE;

			8:
				Out4 := TRUE;

			9:
				Out1 := TRUE;
				Out4 := TRUE;

			10:
				Out2 := TRUE;
				Out4 := TRUE;

			11:
				Out1 := TRUE;
				Out2 := TRUE;
				Out4 := TRUE;

			12:
				Out3 := TRUE;
				Out4 := TRUE;

			13:
				Out1 := TRUE;
				Out3 := TRUE;
				Out4 := TRUE;

			14:
				Out2 := TRUE;
				Out3 := TRUE;
				Out4 := TRUE;

			15:
				Out1 := TRUE;
				Out2 := TRUE;
				Out3 := TRUE;
				Out4 := TRUE;
		END_CASE

		LearnState := READINGS;

	READINGS:	(* Read "SamplesNr" samples, every 10ms *)
		SampleTMR(IN:=NOT SampleTMR.Q);

		IF SampleTMR.Q THEN
			aLearning[LSamplesCtr] := AdcValue;
			LSamplesCtr := LSamplesCtr + 1;

			IF LSamplesCtr = LSamples THEN
				LSamplesCtr := 1;
				SampleTMR(IN:=FALSE);
				LearnState := SWITCH_OFF;
			END_IF
		END_IF

	SWITCH_OFF:	(* Evaluate reference value *)
		CASE Combination OF

			1:
				Out1 := FALSE;

			2:
				Out2 := FALSE;

			3:
				Out1 := FALSE;
				Out2 := FALSE;

			4:
				Out3 := FALSE;

			5:
				Out1 := FALSE;
				Out3 := FALSE;

			6:
				Out2 := FALSE;
				Out3 := FALSE;

			7:
				Out1 := FALSE;
				Out2 := FALSE;
				Out3 := FALSE;

			8:
				Out4 := FALSE;

			9:
				Out1 := FALSE;
				Out4 := FALSE;

			10:
				Out2 := FALSE;
				Out4 := FALSE;

			11:
				Out1 := FALSE;
				Out2 := FALSE;
				Out4 := FALSE;

			12:
				Out3 := FALSE;
				Out4 := FALSE;

			13:
				Out1 := FALSE;
				Out3 := FALSE;
				Out4 := FALSE;

			14:
				Out2 := FALSE;
				Out3 := FALSE;
				Out4 := FALSE;

			15:
				Out1 := FALSE;
				Out2 := FALSE;
				Out3 := FALSE;
				Out4 := FALSE;
		END_CASE

		(* Reference value is the mean value of the measured samples *)
		Lux_ref[ID, Combination] := MEAN_VALUE(ADR(aLearning), LSamples);
		(* Reset readings array *)
		RESET_ARRAY(pData:=ADR(aLearning), Size:=LSamples);

		Combination := Combination + 1;

		IF Combination < EXPT(2,Lines) THEN
			LearnState := SWITCH_ON;
		ELSE
			Combination := 1;
			Status := NORMAL_STATE;			(* Back to wait state *)
		END_IF
END_CASE
END_ACTION
ACTION Measure:
(* Proceed with measure only if not in learning mode *)
IF Status=NORMAL_STATE THEN
	(* If window is full (number of samples as required) go on with mean value e check threshold *)
	IF MSamplesCtr=MSamples THEN

		SHIFT_ARRAY(pData:=ADR(aReading), Size:=MSamples);
		aReading[MSamples] := AdcValue;

		ReadValue := MEAN_VALUE(ADR(aReading), MSamples);
		CheckThreshold();

	ELSE
		(* Window is not full, keep going filling in samples before make a check *)
		aReading[MSamplesCtr] := AdcValue;
		MSamplesCtr := MSamplesCtr + 1;

	END_IF
END_IF
END_ACTION

(* POU Plant_Objects/obj_CRON, ST *)
FUNCTION_BLOCK obj_CRON
(* === CRONOGRAFO STANDARD ===
   v1.0[16/04/15] - Versioning
   v1.1[19/05/15] - Removed DB creation from previous year
*)
VAR_INPUT
	(* Settings *)
	ID			: BYTE;		(* Index of instanced object *)

	InitOK		: BOOL;
	Alarm		: BOOL;
	Warning		: BOOL;

	Profile		: typ_Cron_Profile; 				(* Profilo attivo *)
	ProfileNr	: BYTE;								(* Indice profilo attivo *)
	CalendarIdx : WORD;								(* Indice calendario attivo *)
	Jolly		: ARRAY[0..9] OF typ_Cron_Jolly;	(* Jolly attivi *)

END_VAR
VAR_IN_OUT
END_VAR
VAR_OUTPUT
	SetPoint		: INT;
	(* Status *)
	Status_Log		: BYTE;
	Status_Vis 		: DWORD;
END_VAR
VAR
	Buf: 	ARRAY[0..512] OF BYTE; (* AVOID THIS!! *)
	hFile: 	DWORD;
	sFile: 	STRING;
	sFile2: STRING;

	i:		WORD;
	t1:		DWORD;
	t2:		BOOL;

END_VAR
(* Check initialization *)
IF NOT InitOK THEN Init(); END_IF

(* Chrono *)
IF CalendarIdx<>Sys.Time_CT_Day THEN DB_Load(); END_IF
SetPoint:=Profile.Setpoint[Sys.Time_CT_Quarter];

(* Check jolly *)
FOR i := 0 TO 9 DO
	IF ( DT_TO_DWORD(Jolly[i].Start)>0  AND Jolly[i].End>Jolly[i].Start AND
	     Jolly[i].Start<=Sys.Time_CT_DT AND Jolly[i].End>Sys.Time_CT_DT ) THEN
			SetPoint:=Jolly[i].Temp;
	END_IF
END_FOR


(* Status color *)
   IF Alarm   THEN Status_Log:=2; Status_Vis:=COLOR_RED;
ELSIF Warning THEN Status_Log:=1; Status_Vis:=COLOR_YELLOW;
              ELSE Status_Log:=0; Status_Vis:=COLOR_GREEN;
			  END_IF
END_FUNCTION_BLOCK
ACTION DB_Create:
(*
(* Check presence of previous year *)
sFile2:=REPLACE(STR1:=sFile, STR2:=WORD_TO_STRING(Sys.Time_Year-1), L:=4, P:=LEN(FilesPath)+1);
hFile:=SysFileOpen(FileName:=sFile2, Mode:='r');
IF hFile<>0 THEN
	(* Check file version and close *)
	SysFileRead(File:=hFile, Buffer:=ADR(Buf), Size:=1);
	SysFileClose(File:=hFile);
END_IF
IF hFile<>0 AND Buf[0]=1 THEN
	(* Copy file *)
	SysFileCopy(FileDest:=sFile, FileSource:=sFile2);
ELSE
*)
	(* Create empty file *)
	hFile:=SysFileOpen(FileName:=sFile, Mode:='w');

	MEMCLR(pDestinationAddress:=ADR(Buf), BytesToClear:=SIZEOF(Buf));
	FOR i := 0 TO 10239 BY 512 DO
		t1:=SysFileWrite(File:=hFile, Buffer:=ADR(Buf), Size:=512);
	END_FOR
	Buf[0]:=1;
	t2:=SysFileSetPos(File:=hFile, Pos:=0);
	t1:=SysFileWrite(File:=hFile, Buffer:=ADR(Buf), Size:=1);
	SysFileClose(File:=hFile);
(*
END_IF
*)
END_ACTION
ACTION DB_Load:
DB_SetName();

(* Open data file *)
hFile:=SysFileOpen(FileName:=sFile, Mode:='r');

(* File not found *)
IF hFile=0 THEN
	Warning:=TRUE;
	LogEv(EL_Wrn,EO_CRON,ID,1,'No_data_file');
	DB_Create();
	(* Reopen file *)
	hFile:=SysFileOpen(FileName:=sFile, Mode:='r');
	IF hfile=0 THEN
		Alarm:=TRUE;
		LogEv(EL_Alarm,EO_CRON,ID,3,'Filesystem_error');
		RETURN;
	END_IF
END_IF

(* Check version *)
SysFileRead(File:=hFile, Buffer:=ADR(Buf), Size:=1);
IF Buf[0]<>1 THEN
	IF NOT Alarm THEN
		Alarm:=TRUE;
		LogEv(EL_Alarm,EO_CRON,ID,2,'Bad_data_version');
	END_IF
	SysFileClose(File:=hFile);
	RETURN;
END_IF

(* Read Jolly data *)
t2:=SysFileSetPos(File:=hFile, Pos:=512);
t1:=SysFileRead(File:=hFile, Buffer:=ADR(Jolly), Size:=SIZEOF(Jolly));
(* Read active profile index *)
CalendarIdx:=Sys.Time_CT_Day;
t2:=SysFileSetPos(File:=hFile, Pos:=(1024+4*CalendarIdx));
t1:=SysFileRead(File:=hFile, Buffer:=ADR(ProfileNr), Size:=SIZEOF(ProfileNr));
(* Read active profile *)
t2:=SysFileSetPos(File:=hFile, Pos:=(3072+512*ProfileNr));
t1:=SysFileRead(File:=hFile, Buffer:=ADR(Profile), Size:=SIZEOF(Profile));

(* Close file and validate data *)
SysFileClose(File:=hFile);
END_ACTION
ACTION DB_SetName:
(* Create current filename 'yyyyCRnn.DAT' *)
sFile:=CONCAT(FilesPath,WORD_TO_STRING(Sys.Time_Year));
sFile:=CONCAT(STR1:=sFile, STR2:='CR');
IF ID<10 THEN
sFile:=CONCAT(STR1:=sFile, STR2:='0');
END_IF
sFile:=CONCAT(STR1:=sFile, STR2:=BYTE_TO_STRING(ID));
sFile:=CONCAT(STR1:=sFile, STR2:='.DAT');
END_ACTION
ACTION Init:
DB_Load();
InitOK:=TRUE;
END_ACTION

(* POU Plant_Objects/obj_CRON_EDITOR, ST *)
FUNCTION_BLOCK obj_CRON_EDITOR
(* === EDITOR CRONOGRAFO ===
   v1.0[16/04/15] - Versioning
   v1.1[19/05/15] - Create empty profile when not found
*)
VAR_INPUT

	(* Common selections *)
	CN_Sel:			BYTE:=1;
	CN_Act:			BYTE;
	CN_YSel:		WORD:=2015;
	CN_YAct:		WORD;

	(* Profile editor *)
	PR_Sel: 		BYTE:=1;
	PR_Act:			BYTE;
	PR_TT:			REAL;
	PR:				typ_Cron_Profile;
	(* Profile signals *)
	PR_Load:		BOOL;
	PR_Save:		BOOL;

	(* Calendar editor *)
	CA_Sel:			BYTE:=1; (* Calendar month selected *)
	CA_Act:			BYTE;    (* Calendar month active *)
	CA_DayF:		BYTE:=0;
	CA_DayL:		BYTE:=31;
	CA_TPR:			BYTE;
	CA:				typ_Cron_Calendar; (* Only used for first 32 entries *)
	(* Calendar signals *)
	CA_Load:		BOOL;
	CA_Save:		BOOL;

	(* Jolly editor *)
	JL:				ARRAY[0..9] OF typ_Cron_Jolly;
	(* Jolly signals *)
	JL_Load:		BOOL;
	JL_Save:		BOOL;

END_VAR
VAR_OUTPUT
	Message		: STRING;
END_VAR
VAR
	sFileName	: STRING;
	sFileMode	: STRING;
	hFile		: DWORD;
	Buf			: ARRAY[0..512] OF BYTE; (* AVOID THIS!! *)

	i			: WORD;
	ver			: BYTE;
	r1			: BOOL;
	r2			: DWORD;

END_VAR
IF PR_Load THEN PR_Load_Exe(); PR_Load:=FALSE; END_IF
IF PR_Save THEN PR_Save_Exe(); PR_Save:=FALSE; END_IF
IF CA_Load THEN CA_Load_Exe(); CA_Load:=FALSE; END_IF
IF CA_Save THEN CA_Save_Exe(); CA_Save:=FALSE; END_IF
IF JL_Load THEN JL_Load_Exe(); JL_Load:=FALSE; END_IF
IF JL_Save THEN JL_Save_Exe(); JL_Save:=FALSE; END_IF
END_FUNCTION_BLOCK
ACTION CA_Load_Exe:
sFileMode:='r';
FileOpen();

IF hFile<>0 THEN

	(* Read calendar month *)
	FOR i := 0 TO 31 DO
		r1:=SysFileSetPos(File:=hFile, Pos:=(1024 + ((CA_Sel-1)*32 + i)*4));
		r2:=SysFileRead(File:=hFile, Buffer:=ADR(CA.Profile[i]), Size:=1);
	END_FOR

	(* Close file *)
	SysFileClose(File:=hFile);

	(* Validate data *)
	CA_Act :=CA_Sel;
	CN_Act :=CN_Sel;
	CN_YAct:=CN_YSel;

	Message:='Calendar load OK';

END_IF
END_ACTION
ACTION CA_Save_Exe:
sFileMode:='a';
FileOpen();

IF hFile<>0 THEN

	(* Write calendar month *)
	FOR i := 0 TO 31 DO
		r1:=SysFileSetPos(File:=hFile, Pos:=(1024 + ((CA_Sel-1)*32 + i)*4));
		r2:=SysFileGetPos(hFile);
		r2:=SysFileWrite(File:=hFile, Buffer:=ADR(CA.Profile[i]), Size:=1);
	END_FOR

	(* Close file *)
	SysFileClose(File:=hFile);

	Message:='Calendar save OK';

END_IF
END_ACTION
ACTION FileOpen:
(* Create current filename 'yyyyCRnn.DAT' *)
sFileName:=CONCAT(FilesPath,WORD_TO_STRING(CN_YSel));
sFileName:=CONCAT(STR1:=sFileName, STR2:='CR');
IF CN_Sel<10 THEN
sFileName:=CONCAT(STR1:=sFileName, STR2:='0');
END_IF
sFileName:=CONCAT(STR1:=sFileName, STR2:=BYTE_TO_STRING(CN_Sel));
sFileName:=CONCAT(STR1:=sFileName, STR2:='.DAT');

(* Check file version and size! *)
(* ... *)

(* Open data file *)
hFile:=SysFileOpen(FileName:=sFileName, Mode:='r');

(* File not found *)
IF hFile=0 THEN
	Message:='File not found - created empty file';
	(* Create empty file *)
	hFile:=SysFileOpen(FileName:=sFileName, Mode:='w');
	MEMCLR(pDestinationAddress:=ADR(Buf), BytesToClear:=SIZEOF(Buf));
	FOR i := 0 TO 10239 BY 512 DO
		SysFileWrite(File:=hFile, Buffer:=ADR(Buf), Size:=512);
	END_FOR
	Buf[0]:=1;
	SysFileSetPos(File:=hFile, Pos:=0);
	SysFileWrite(File:=hFile, Buffer:=ADR(Buf), Size:=1);
END_IF

(* Close file *)
SysFileClose(File:=hFile);

(* Open data file *)
hFile:=SysFileOpen(FileName:=sFileName, Mode:=sFileMode);
END_ACTION
ACTION JL_Load_Exe:
sFileMode:='r';
FileOpen();

IF hFile<>0 THEN

	(* Read jolly *)
	r1:=SysFileSetPos(File:=hFile, Pos:=512);
	r2:=SysFileRead(File:=hFile, Buffer:=ADR(JL), Size:=SIZEOF(JL));

	(* Close file *)
	SysFileClose(File:=hFile);

	(* Validate data *)
	CN_Act:=CN_Sel;
	CN_YAct:=CN_YSel;

	Message:='Jolly load OK';

END_IF
END_ACTION
ACTION JL_Save_Exe:
sFileMode:='a';
FileOpen();

IF hFile<>0 THEN

	(* Write selected profile *)
	r1:=SysFileSetPos(File:=hFile, Pos:=512);
	r2:=SysFileWrite(File:=hFile, Buffer:=ADR(JL), Size:=SIZEOF(JL));

	(* Close file *)
	SysFileClose(File:=hFile);

	Message:='Jolly save OK';

END_IF
END_ACTION
ACTION PR_Load_Exe:
sFileMode:='r';
FileOpen();

IF hFile<>0 THEN

	(* Read selected profile *)
	r1:=SysFileSetPos(File:=hFile, Pos:=(3072 + 512*PR_Sel));
	r2:=SysFileRead(File:=hFile, Buffer:=ADR(PR), Size:=SIZEOF(PR));

	(* Close file *)
	SysFileClose(File:=hFile);

	(* Validate data *)
	PR_Act:=PR_Sel;
	CN_Act:=CN_Sel;
	CN_YAct:=CN_YSel;

	Message:='Profile load OK';

END_IF
END_ACTION
ACTION PR_Save_Exe:
sFileMode:='a';
FileOpen();

IF hFile<>0 THEN

	(* Write selected profile *)
	r1:=SysFileSetPos(File:=hFile, Pos:=(3072 + 512*PR_Sel));
	r2:=SysFileWrite(File:=hFile, Buffer:=ADR(PR), Size:=SIZEOF(PR));

	(* Close file *)
	SysFileClose(File:=hFile);

	Message:='Profile save OK';

END_IF
END_ACTION

(* POU Plant_Objects/obj_HVAC_LENNOX_FGK190H2M, ST *)
FUNCTION_BLOCK obj_HVAC_LENNOX_FGK190H2M
VAR_INPUT
	(* Var globale per il mondo *)

	(* Settings *)
	ID						: BYTE;
	ADDRESS					: BYTE:=31;
	Refresh_Period			: TIME:=t#3m;
	(* Controls *)
	Refresh_Auto			: BOOL:=TRUE; (* Enable automatic refresh *)
	Refresh_Now				: BOOL; 	  (* Force an immediate refresh *)

	Heartbeat				:WORD;	(*holding registers 1 *)
	SP_Raffreddamento		:WORD;	(*holding registers 2 *)
	SP_Riscaldamento		:WORD;	(*holding registers 3 *)


	TempAmbienteBMS			:WORD;	(*holding registers 20 *)
	UmiditaAmbienteBMS		:WORD;	(*holding registers 21 *)
	TempEsternaBMS			:WORD;	(*holding registers 22 *)
	UmiditaEsternaBMS		:WORD;	(*holding registers 23 *)

	On_Off_Unita			:WORD;    (* holding registers  84 *)

	SP_MinPortataAriaECO	:WORD;	(*holding registers 187 *)
	SP_MAXPortataAriaECO	:WORD;	(*holding registers 188 *)


END_VAR
VAR_IN_OUT
	MODBUS			: obj_MODBUS;
END_VAR
VAR_OUTPUT
	(* Sono read-only tetto il mondo *)

	Data			: typ_MODBUS_HVAC_LENNOX_FGK190H2M_new;
	(* Status *)
	Status_Log		: BYTE;
	Status_Vis 		: DWORD;

END_VAR
VAR

	dly 	 : TON := (PT:=t#5s);
	sta		 : BYTE; 	(* Status *)
	retry	 : BYTE;

	StatoMW: ARRAY [1..8] OF WORD;
	h_Compressore2_h: BOOL;
END_VAR
CASE sta OF
	0: (* === Wait update signals *)
		dly(IN:=NOT (dly.Q OR Refresh_Now OR (NOT Refresh_Auto)));
		IF dly.Q OR Refresh_Now THEN
			dly.PT:=Refresh_Period;
			Refresh_Now:=FALSE;
			sta:=1;
		END_IF

	1: (* === Start update when MB is free *)
		IF NOT (MODBUS.MB_Lock OR MODBUS.MB_Start) THEN
			MODBUS.MB_Lock:=TRUE;
			MODBUS.MB_Query.SlaveAddress:=ADDRESS;

			(* Start query *)
			MODBUS.MB_Query.FunctionCode		:=16#03;
			MODBUS.MB_Query.Read_StartAddress	:=16#24; (* Leggo le varibili da loggare chiamate Analogiche dal registro 36 *)
			MODBUS.MB_Query.Read_Quantity		:=16#0F;

			MODBUS.MB_Start:=TRUE;
			sta:=2;
	END_IF


(* Leggo le varibili da loggare chiamate Analogiche dal registro 36 *)
	2:	IF NOT MODBUS.MB_Start THEN
			IF MODBUS.MB_MASTER.MB_Error<>MB_NO_ERROR OR MODBUS.MB_Resp.Error<>0 THEN
				sta:=100;
			ELSE



				(* Read response data *)
				Data.ErrorCode:= (MODBUS.MB_Resp.Data[ 0]);
				Data.TempAmbiente:=WORD_TO_INT(MODBUS.MB_Resp.Data[ 2]);
				Data.TempEserno:=WORD_TO_INT(MODBUS.MB_Resp.Data[ 4]);
				Data.TempMandata:=WORD_TO_INT(MODBUS.MB_Resp.Data[ 5]);
				Data.TempRipresa:=WORD_TO_INT(MODBUS.MB_Resp.Data[ 8]);
				Data.RelUmiditaAmbiente:=WORD_TO_INT(MODBUS.MB_Resp.Data[ 10]);
				Data.AbsUmiditaAmbiente:=WORD_TO_INT(MODBUS.MB_Resp.Data[12]);
				Data.RelUmiditaEsterno:=WORD_TO_INT(MODBUS.MB_Resp.Data[14]);
				Data.AbsUmiditaEsterno:=WORD_TO_INT(MODBUS.MB_Resp.Data[16]);
				Data.PressDiff:=WORD_TO_INT(MODBUS.MB_Resp.Data[18]);
				Data.ApValvAria:=WORD_TO_INT(MODBUS.MB_Resp.Data[22]);
				Data.ApValvGAS:=WORD_TO_INT(MODBUS.MB_Resp.Data[24]);
				Data.ResElettrica:=WORD_TO_INT(MODBUS.MB_Resp.Data[26]);
				Data.PercUmidificatore:=WORD_TO_INT(MODBUS.MB_Resp.Data[28]);

				(* Start query *)
				MODBUS.MB_Query.Read_StartAddress:=16#3E;
				MODBUS.MB_Query.Read_Quantity:=16#16;
				MODBUS.MB_Start:=TRUE;
				sta:=3;
			END_IF
		END_IF

(* Leggo le varibili da loggare chiamatecontatori tempo funzionament  dal registro 62 *)
	3:	IF NOT MODBUS.MB_Start THEN
			IF MODBUS.MB_MASTER.MB_Error<>MB_NO_ERROR OR MODBUS.MB_Resp.Error<>0 THEN
				sta:=100;
			ELSE
				(* Read response data *)
				Data.h_VentSoffiante := ((MODBUS.MB_Resp.Data[ 1])* 65536)+MODBUS.MB_Resp.Data[ 0];
				Data.h_Compressore1 := ((MODBUS.MB_Resp.Data[ 3])* 65536)+MODBUS.MB_Resp.Data[ 2];
				Data.h_Compressore2 := ((MODBUS.MB_Resp.Data[ 5])* 65536)+MODBUS.MB_Resp.Data[ 4];
				Data.h_Compressore3 := ((MODBUS.MB_Resp.Data[ 7])* 65536)+MODBUS.MB_Resp.Data[ 6];
				Data.h_Compressore4 := ((MODBUS.MB_Resp.Data[ 9])* 65536)+MODBUS.MB_Resp.Data[ 8];

				(* Start query *)

				MODBUS.MB_Query.FunctionCode:=16#03;
				MODBUS.MB_Query.Read_StartAddress:=16#4A;   (* Leggo lo stato degli allarmi 74 *)
				MODBUS.MB_Query.Read_Quantity:=16#10;
				MODBUS.MB_Start:=TRUE;
				sta:=4;
			END_IF
		END_IF
(* Leggo lo stato degli allarmi *)
	4:	IF NOT MODBUS.MB_Start THEN
			IF MODBUS.MB_MASTER.MB_Error<>MB_NO_ERROR OR MODBUS.MB_Resp.Error<>0 THEN
				sta:=100;
			ELSE
				(* Read response data *)
				Data.bit_Allarme01:=(MODBUS.MB_Resp.Data[ 0]);
				Data.bit_Allarme02:=(MODBUS.MB_Resp.Data[ 1]);
				Data.bit_Allarme03:=(MODBUS.MB_Resp.Data[ 2]);
				Data.bit_Allarme04:=(MODBUS.MB_Resp.Data[ 3]);
				Data.bit_Allarme05:=(MODBUS.MB_Resp.Data[ 4]);
				Data.bit_Allarme06:=(MODBUS.MB_Resp.Data[ 5]);
				Data.bit_Allarme07:=(MODBUS.MB_Resp.Data[ 6]);



			(* Verifico la presenza di nuovi allarmi ed eventualemte Loggo l'evento *)


				IF 	(Data.bit_Allarme01>StatoMW[1] ) OR  (Data.bit_Allarme02>StatoMW[2] ) OR
					(Data.bit_Allarme03>StatoMW[3] ) OR  (Data.bit_Allarme04>StatoMW[4] ) OR
					(Data.bit_Allarme05>StatoMW[5] ) OR  (Data.bit_Allarme06>StatoMW[6] ) OR
					(Data.bit_Allarme07>StatoMW[7] )  THEN
					LogEv(EL_Log,EO_ANZ,ID,3,WORD_TO_STRING(Data.ErrorCode));
				ELSE
					StatoMW[1]:= Data.bit_Allarme01;
					StatoMW[2]:= Data.bit_Allarme02;
					StatoMW[3]:= Data.bit_Allarme03;
					StatoMW[4]:= Data.bit_Allarme04;
					StatoMW[5]:= Data.bit_Allarme05;
					StatoMW[6]:= Data.bit_Allarme06;
					StatoMW[7]:= Data.bit_Allarme07;
				END_IF
				sta:=10;
			END_IF
		END_IF

(* scrivo i controlli  *)

10:
		IF NOT (MODBUS.MB_Lock OR MODBUS.MB_Start) THEN
			MODBUS.MB_Query.SlaveAddress:=ADDRESS;


				MODBUS.MB_Query.Write_Data[0]:=Heartbeat;    					(* questa varibile deve essere sempre aggiornata a 300 è il Heartbeat  *)
				MODBUS.MB_Query.Write_Data[1]:=SP_Raffreddamento;   		(* SP_Raffreddamento			:WORD;	(*holding registers 2 *)  *)
				MODBUS.MB_Query.Write_Data[2]:=SP_Riscaldamento; 			(* SP_Riscaldamento				:WORD;	(*holding registers 3 *)  *)

				(* Start query *)
				MODBUS.MB_Query.FunctionCode:=16#10;
				MODBUS.MB_Query.Read_StartAddress:=16#0; (*Scrivo le Variabili al registro 0 *)
				MODBUS.MB_Query.Read_Quantity:=16#4;
				MODBUS.MB_Start:=TRUE;
				sta:=11;

		END_IF

	11:	IF NOT MODBUS.MB_Start THEN
			IF MODBUS.MB_MASTER.MB_Error<>MB_NO_ERROR OR MODBUS.MB_Resp.Error<>0 THEN
				sta:=100;
			ELSE


				MODBUS.MB_Query.Write_Data[0]:=TempAmbienteBMS;    					(* TempAmbienteBMS			:WORD;	(*holding registers 20 *)  *)
				MODBUS.MB_Query.Write_Data[1]:=UmiditaAmbienteBMS;   					(* UmiditaAmbienteBMS			:WORD;	(*holding registers 21 *)  *)
				MODBUS.MB_Query.Write_Data[2]:=TempEsternaBMS; 					(* TempEsternaBMS				:WORD;	(*holding registers 22 *) *)
				MODBUS.MB_Query.Write_Data[3]:=UmiditaEsternaBMS; 					(* UmiditaEsternaBMS			:WORD;	(*holding registers 23 *) *)

				(* Start query *)
				MODBUS.MB_Query.FunctionCode:=16#10;
				MODBUS.MB_Query.Read_StartAddress:=16#14; (*Scrivo le Variabili al registro 20 *)
				MODBUS.MB_Query.Read_Quantity:=16#6;
				MODBUS.MB_Start:=TRUE;
				sta:=12;
			END_IF
		END_IF

	12:	IF NOT MODBUS.MB_Start THEN
			IF MODBUS.MB_MASTER.MB_Error<>MB_NO_ERROR OR MODBUS.MB_Resp.Error<>0 THEN
				sta:=100;
			ELSE


				MODBUS.MB_Query.Write_Data[0]:=On_Off_Unita;    					(* On_Off_Unita					:WORD;    (* holding registers  84 *)  *)
				MODBUS.MB_Query.Write_Data[1]:=0;
				MODBUS.MB_Query.Write_Data[2]:=0;
				MODBUS.MB_Query.Write_Data[3]:=0;

				(* Start query *)
				MODBUS.MB_Query.FunctionCode:=16#10;
				MODBUS.MB_Query.Read_StartAddress:=16#54; (*Scrivo le Variabili al registro 84 *)
				MODBUS.MB_Query.Read_Quantity:=16#6;
				MODBUS.MB_Start:=TRUE;
				sta:=13;
			END_IF
		END_IF

	13:	IF NOT MODBUS.MB_Start THEN
			IF MODBUS.MB_MASTER.MB_Error<>MB_NO_ERROR OR MODBUS.MB_Resp.Error<>0 THEN
				sta:=100;
			ELSE


				MODBUS.MB_Query.Write_Data[0]:=SP_MinPortataAriaECO;    	(* On_Off_Unita					:WORD;    (* holding registers  84 *)  *)
				MODBUS.MB_Query.Write_Data[1]:=SP_MAXPortataAriaECO;
				MODBUS.MB_Query.Write_Data[2]:=0;
				MODBUS.MB_Query.Write_Data[3]:=0;

				(* Start query *)
				MODBUS.MB_Query.FunctionCode:=16#10;
				MODBUS.MB_Query.Read_StartAddress:=16#BB; (*Scrivo le Variabili al registro 187 *)
				MODBUS.MB_Query.Read_Quantity:=16#6;
				MODBUS.MB_Start:=TRUE;
				sta:=14;
			END_IF
		END_IF


	14:	IF NOT MODBUS.MB_Start THEN
			IF MODBUS.MB_MASTER.MB_Error<>MB_NO_ERROR OR MODBUS.MB_Resp.Error<>0 THEN
				sta:=100;
			ELSE
				MODBUS.MB_Lock:=FALSE;
				sta:=0;
			END_IF
		END_IF






	100: (* === Check MODBUS error *)
			(* Release MODBUS *)
			MODBUS.MB_Lock:=FALSE;
			(* Retries *)
			retry:=retry+1;
			IF retry>3 THEN
				retry:=0;
				(* Signal event *)
				IF Status_Log<>2 THEN
					LogEv(EL_Alarm,EO_HVAC,ID,2,'');
				END_IF
				(* Update status *)
				Status_Log:=2;
				Status_Vis:=COLOR_RED;
			END_IF
			sta:=0;

ELSE
	sta:=0;
END_CASE
END_FUNCTION_BLOCK
ACTION AddLogData:
Logger.s1:=INSERT('&HVAC=',BYTE_TO_STRING(ID),4);
IF ID<10 THEN Logger.s1:=INSERT(Logger.s1,'0',4); END_IF

Logger.s1:=CONCAT(Logger.s1,INT_TO_STRING(Data.TempMandata));			Logger.s1:=CONCAT(Logger.s1,';');
Logger.s1:=CONCAT(Logger.s1,INT_TO_STRING(Data.TempRipresa));			Logger.s1:=CONCAT(Logger.s1,';');
Logger.s1:=CONCAT(Logger.s1,INT_TO_STRING(Data.PressDiff));				Logger.s1:=CONCAT(Logger.s1,';');
Logger.s1:=CONCAT(Logger.s1,INT_TO_STRING(Data.ApValvAria));			Logger.s1:=CONCAT(Logger.s1,';');
Logger.s1:=CONCAT(Logger.s1,INT_TO_STRING(Data.ApValvGAS));				Logger.s1:=CONCAT(Logger.s1,';');
Logger.s1:=CONCAT(Logger.s1,INT_TO_STRING(Data.ResElettrica));			Logger.s1:=CONCAT(Logger.s1,';');
Logger.s1:=CONCAT(Logger.s1,INT_TO_STRING(Data.ApValvAcquaCalda));		Logger.s1:=CONCAT(Logger.s1,';');
Logger.s1:=CONCAT(Logger.s1,INT_TO_STRING(Data.PercUmidificatore));		Logger.s1:=CONCAT(Logger.s1,';');

(* Mancano bit allarmi/stato	*)

Logger.s1:=CONCAT(Logger.s1,DWORD_TO_STRING(Data.h_VentSoffiante));		Logger.s1:=CONCAT(Logger.s1,';');
Logger.s1:=CONCAT(Logger.s1,DWORD_TO_STRING(Data.h_Compressore1));		Logger.s1:=CONCAT(Logger.s1,';');
Logger.s1:=CONCAT(Logger.s1,DWORD_TO_STRING(Data.h_Compressore2));		Logger.s1:=CONCAT(Logger.s1,';');
Logger.s1:=CONCAT(Logger.s1,DWORD_TO_STRING(Data.h_Compressore3));		Logger.s1:=CONCAT(Logger.s1,';');
Logger.s1:=CONCAT(Logger.s1,DWORD_TO_STRING(Data.h_Compressore4));		Logger.s1:=CONCAT(Logger.s1,';');






Logger.s1:=CONCAT(Logger.s1,WORD_TO_STRING(Data.ErrorCode));			Logger.s1:=CONCAT(Logger.s1,';');
Logger.s1:=CONCAT(Logger.s1,INT_TO_STRING(Data.TempAmbiente));			Logger.s1:=CONCAT(Logger.s1,';');
Logger.s1:=CONCAT(Logger.s1,INT_TO_STRING(Data.TempEserno));			Logger.s1:=CONCAT(Logger.s1,';');
Logger.s1:=CONCAT(Logger.s1,INT_TO_STRING(Data.RelUmiditaAmbiente));		Logger.s1:=CONCAT(Logger.s1,';');
Logger.s1:=CONCAT(Logger.s1,INT_TO_STRING(Data.AbsUmiditaAmbiente));		Logger.s1:=CONCAT(Logger.s1,';');
Logger.s1:=CONCAT(Logger.s1,INT_TO_STRING(Data.RelUmiditaEsterno));			Logger.s1:=CONCAT(Logger.s1,';');
Logger.s1:=CONCAT(Logger.s1,INT_TO_STRING(Data.AbsUmiditaEsterno));		Logger.s1:=CONCAT(Logger.s1,';');
Logger.s1:=CONCAT(Logger.s1,INT_TO_STRING(Data.LivCO2));					Logger.s1:=CONCAT(Logger.s1,';');
Logger.s1:=CONCAT(Logger.s1,WORD_TO_STRING(Data.bit_Allarme01));		Logger.s1:=CONCAT(Logger.s1,';');
Logger.s1:=CONCAT(Logger.s1,WORD_TO_STRING(Data.bit_Allarme02));		Logger.s1:=CONCAT(Logger.s1,';');
Logger.s1:=CONCAT(Logger.s1,WORD_TO_STRING(Data.bit_Allarme03));		Logger.s1:=CONCAT(Logger.s1,';');
Logger.s1:=CONCAT(Logger.s1,WORD_TO_STRING(Data.bit_Allarme04));		Logger.s1:=CONCAT(Logger.s1,';');
Logger.s1:=CONCAT(Logger.s1,WORD_TO_STRING(Data.bit_Allarme05));		Logger.s1:=CONCAT(Logger.s1,';');
Logger.s1:=CONCAT(Logger.s1,WORD_TO_STRING(Data.bit_Allarme06));		Logger.s1:=CONCAT(Logger.s1,';');
Logger.s1:=CONCAT(Logger.s1,WORD_TO_STRING(Data.bit_Allarme07));		Logger.s1:=CONCAT(Logger.s1,';');


Logger.s1:=CONCAT(Logger.s1,BYTE_TO_STRING(Status_Log));
ADDSTRING(ADR(Logger.TData), ADR(Logger.s1), Logger.TLen);
END_ACTION

(* POU Plant_Objects/obj_MODBUS, ST *)
FUNCTION_BLOCK obj_MODBUS
(* === MODBUS PROTOCOL INTERFACE ===
   v1.1[19/06/15] - Added new VARS allocation and searching
*)
VAR CONSTANT
	VARS_Max	: BYTE := 32;
END_VAR
VAR_INPUT
	(* Settings *)
	ID			: BYTE;
	COM			: BYTE;
	BAUDRATE	: COM_BAUDRATE;
	RS485		: BOOL := FALSE;

	(* Interface *)
	MB_MASTER	: MODBUS_EXTENDED_MASTER;
	MB_Start	: BOOL;
	MB_Query	: typModbusExtendedQuery;
	MB_Resp		: typModbusResponse;
	MB_Lock		: BOOL;

	(* Variables management *)
	VARS_En		: BOOL;
	VARS		: ARRAY [0..VARS_Max] OF typ_MODBUS_VAR;
	VARS_Check	: BOOL;
	VARS_Alarm	: BOOL;

	(* Variables allocation *)
	VAR_Pointer : POINTER TO ARRAY[0..99] OF WORD;
	VAR_Cfg		: POINTER TO typ_MODBUS_VAR;
END_VAR
VAR_OUTPUT
	(* Status *)
	Status_Log	: BYTE;
	Status_Vis	: DWORD;
END_VAR
VAR
	sta         : BYTE :=0;
	i			: BYTE;
	j			: BYTE;
	Alarm		: FLT_EVENT;

	VarTmr		: TON := (PT:=T#1s);
	VarSta		: BYTE; (* Status *)
	VarCnt		: BYTE; (* Scan counter *)
	VarRetry	: BYTE;
	VarAlarm	: BYTE; (* Last variable with errors *)
END_VAR
(* NB: Timeout has been changed: 750ms instead of 250ms as usual. This because Frer declares
       "Minimum response time-out (to be set on the master): 500ms." 		*)
MB_MASTER(ENABLE:=TRUE,	ASCII_Mode:=FALSE, bCOM_PORT:=COM, cbCOM_BAUDRATE:=BAUDRATE, cpCOM_PARITY:=PARITY_NO,
		csCOM_STOPBITS:=STOPBITS_2,	cbsCOM_BYTESIZE:=BS_8, cfCOM_FLOW_CONTROL:=SEL(RS485,NO_FLOW_CONTROL,HALFDUPLEX),
		tTIME_OUT:=t#250ms,	StartFunction:=MB_Start, ExtQuery:=MB_Query, Response:=MB_Resp);

(* Process variable management *)
IF VARS_En THEN VARS_Process(); END_IF

(* Check status *)
Alarm(IN:=(MB_MASTER.bInterfaceError<>0));
IF Alarm.EVH THEN
	LogEv(SEL(MB_MASTER.bInterfaceError<>3,EL_Wrn,EL_Alarm),EO_MODBUS,ID,1,BYTE_TO_STRING(MB_MASTER.bInterfaceError));
END_IF
IF Alarm.EVL THEN								(* Trigger a fall edge: MODBUS back working *)
	LogEv(EL_Log,EO_MODBUS,ID,2,'MODBUS_OK');
END_IF

(* Log/visu status *)
   IF Alarm.IN   THEN Status_Log:=2; Status_Vis:=COLOR_RED;
ELSIF Vars_Alarm THEN Status_Log:=1; Status_Vis:=COLOR_YELLOW;
  				 ELSE Status_Log:=0; Status_Vis:=COLOR_GREEN;
END_IF
END_FUNCTION_BLOCK
ACTION VAR_Search:
(* Search VAR with specific pointer if not found return first free VAR
	[Last VAR is not active... used as safe area...] 
*)
j:=VARS_Max;
FOR i := 0 TO VARS_Max-1 DO
	IF VARS[i].Variable=0 AND j>i THEN j:=i; END_IF
	IF VARS[i].Variable=VAR_Pointer THEN
		VAR_Cfg:=ADR(VARS[i]);
		RETURN;
	END_IF
END_FOR
VAR_Cfg:=ADR(VARS[j]);
END_ACTION
ACTION VARS_Process:
(* Update var timers *)
VarTmr(IN:=(NOT VarTmr.Q));
IF VarTmr.Q THEN
	FOR i := 0 TO VARS_Max DO
		IF VARS[i].Refresh_Cnt>0 THEN VARS[i].Refresh_Cnt:=VARS[i].Refresh_Cnt-1; END_IF
	END_FOR
	VARS_Check:=TRUE;
END_IF


(* Process status *)
CASE VarSta OF
	0: (* === Init *)
		VarCnt:=0;
		VarSta:=1;

	1: (* === Wait check signal *)
		IF VARS_Check THEN				(* Decremented "Refresh_Cnt" *)
			VARS_Check:=FALSE;
			VarCnt:=0;
			VarSta:=2;
		END_IF

